# B&R Automation Studio project NAEUL004C00R13L518F00 (part 9)

#### Act_Main_P0200.st
```iecst
(** 2018-12-21 **)
ACTION Act_Main_P0200:
		//Conveyor Direction - SMEMA Arrow Indicator
	IF p_tyNtParamCurr.bUIConvDirRL THEN
		fUIInRtStatHide(ADR(tyP0200OpsGen.tyOps.tyBitmapUSIn.uiRtStat));
		fUIInRtStatHide(ADR(tyP0200OpsGen.tyOps.tyBitmapUSOut.uiRtStat));
		fUIInRtStatHide(ADR(tyP0200OpsGen.tyOps.tyTxtLane.uiRtStat));
		fUIInRtStatHide(ADR(tyP0200OpsGen.tyOps.tyHotspotUSAVSMEMA.uiRtStat));
		fUIInRtStatHide(ADR(tyP0200OpsGen.tyOps.tyBitmapUSAComm.uiRtStat));
		fUIInRtStatHide(ADR(tyP0200OpsGen.tyOps.tyBitmapUSAComm.uiMaskRtStat));

		fUIInRtStatHide(ADR(tyP0200OpsGen.tyUSCommB.tyBitmapUSIn.uiRtStat));
		fUIInRtStatHide(ADR(tyP0200OpsGen.tyUSCommB.tyBitmapUSOut.uiRtStat));
		fUIInRtStatHide(ADR(tyP0200OpsGen.tyUSCommB.tyTxtLane.uiRtStat));
		fUIInRtStatHide(ADR(tyP0200OpsGen.tyUSCommB.tyHotspotUSBVSMEMA.uiRtStat));
		fUIInRtStatHide(ADR(tyP0200OpsGen.tyUSCommB.tyBitmapUSBComm.uiRtStat));
		fUIInRtStatHide(ADR(tyP0200OpsGen.tyUSCommB.tyBitmapUSBComm.uiMaskRtStat));

		fUIInRtStatOff(ADR(tyP0200OpsGen.tyOps.tyBitmapUSIn1.uiRtStat));
		fUIInRtStatOff(ADR(tyP0200OpsGen.tyOps.tyBitmapUSOut1.uiRtStat));
		fUIInRtStatOff(ADR(tyP0200OpsGen.tyOps.tyTxtLane1.uiRtStat));
		//	fUIInRtStatOff(ADR(tyP0200OpsGen.tyOps.tyHotspotUSAVSMEMA1.uiRtStat));
		fUIInRtStatOff(ADR(tyP0200OpsGen.tyOps.tyBitmapUSAComm1.uiRtStat));
		fUIInRtStatOff(ADR(tyP0200OpsGen.tyOps.tyBitmapUSAComm1.uiMaskRtStat));

		fUIInRtStatOff(ADR(tyP0200OpsGen.tyUSCommB.tyBitmapUSIn1.uiRtStat));
		fUIInRtStatOff(ADR(tyP0200OpsGen.tyUSCommB.tyBitmapUSOut1.uiRtStat));
		fUIInRtStatOff(ADR(tyP0200OpsGen.tyUSCommB.tyTxtLane1.uiRtStat));
		//	fUIInRtStatOff(ADR(tyP0200OpsGen.tyUSCommB.tyHotspotUSBVSMEMA1.uiRtStat));
		fUIInRtStatOff(ADR(tyP0200OpsGen.tyUSCommB.tyBitmapUSBComm1.uiRtStat));
		fUIInRtStatOff(ADR(tyP0200OpsGen.tyUSCommB.tyBitmapUSBComm1.uiMaskRtStat));

	ELSE

		fUIInRtStatOff(ADR(tyP0200OpsGen.tyOps.tyBitmapUSIn.uiRtStat));
		fUIInRtStatOff(ADR(tyP0200OpsGen.tyOps.tyBitmapUSOut.uiRtStat));
		fUIInRtStatOff(ADR(tyP0200OpsGen.tyOps.tyTxtLane.uiRtStat));
		//		fUIInRtStatOff(ADR(tyP0200OpsGen.tyOps.tyHotspotUSAVSMEMA.uiRtStat));
		fUIInRtStatOff(ADR(tyP0200OpsGen.tyOps.tyBitmapUSAComm.uiRtStat));
		fUIInRtStatOff(ADR(tyP0200OpsGen.tyOps.tyBitmapUSAComm.uiMaskRtStat));

		fUIInRtStatOff(ADR(tyP0200OpsGen.tyUSCommB.tyBitmapUSIn.uiRtStat));
		fUIInRtStatOff(ADR(tyP0200OpsGen.tyUSCommB.tyBitmapUSOut.uiRtStat));
		fUIInRtStatOff(ADR(tyP0200OpsGen.tyUSCommB.tyTxtLane.uiRtStat));
		//	fUIInRtStatOff(ADR(tyP0200OpsGen.tyUSCommB.tyHotspotUSBVSMEMA.uiRtStat));
		fUIInRtStatOff(ADR(tyP0200OpsGen.tyUSCommB.tyBitmapUSBComm.uiRtStat));
		fUIInRtStatOff(ADR(tyP0200OpsGen.tyUSCommB.tyBitmapUSBComm.uiMaskRtStat));

		fUIInRtStatHide(ADR(tyP0200OpsGen.tyOps.tyBitmapUSIn1.uiRtStat));
		fUIInRtStatHide(ADR(tyP0200OpsGen.tyOps.tyBitmapUSOut1.uiRtStat));
		fUIInRtStatHide(ADR(tyP0200OpsGen.tyOps.tyTxtLane1.uiRtStat));
		fUIInRtStatHide(ADR(tyP0200OpsGen.tyOps.tyHotspotUSAVSMEMA1.uiRtStat));
		fUIInRtStatHide(ADR(tyP0200OpsGen.tyOps.tyBitmapUSAComm1.uiRtStat));
		fUIInRtStatHide(ADR(tyP0200OpsGen.tyOps.tyBitmapUSAComm1.uiMaskRtStat));

		fUIInRtStatHide(ADR(tyP0200OpsGen.tyUSCommB.tyBitmapUSIn1.uiRtStat));
		fUIInRtStatHide(ADR(tyP0200OpsGen.tyUSCommB.tyBitmapUSOut1.uiRtStat));
		fUIInRtStatHide(ADR(tyP0200OpsGen.tyUSCommB.tyTxtLane1.uiRtStat));
		fUIInRtStatHide(ADR(tyP0200OpsGen.tyUSCommB.tyHotspotUSBVSMEMA1.uiRtStat));
		fUIInRtStatHide(ADR(tyP0200OpsGen.tyUSCommB.tyBitmapUSBComm1.uiRtStat));
		fUIInRtStatHide(ADR(tyP0200OpsGen.tyUSCommB.tyBitmapUSBComm1.uiMaskRtStat));

	END_IF

	//Display L to R
	tyP0200OpsGen.tyOps.tyHotspotOpsMagInfo.uiRtStat.0	:= p_tyNtParamCurr.bUIConvDirRL = TRUE;

	tyP0200OpsGen.tyOps.tyTxtMag1Slt.uiRtStat.0 		:= p_tyNtParamCurr.bUIConvDirRL = TRUE;
	tyP0200OpsGen.tyOps.tyTxtMag1Backslash.uiRtStat.0	:= p_tyNtParamCurr.bUIConvDirRL = TRUE;
	tyP0200OpsGen.tyOps.tyNumMag1AvlQty.uiRtStat.0		:= p_tyNtParamCurr.bUIConvDirRL = TRUE;
	tyP0200OpsGen.tyOps.tyNumMag1TtlSlt.uiRtStat.0		:= p_tyNtParamCurr.bUIConvDirRL = TRUE;

	tyP0200OpsGen.tyOps.tyTxtMag2Slt.uiRtStat.0 		:= p_tyNtParamCurr.bUIConvDirRL = TRUE;
	tyP0200OpsGen.tyOps.tyTxtMag2Backslash.uiRtStat.0	:= p_tyNtParamCurr.bUIConvDirRL = TRUE;
	tyP0200OpsGen.tyOps.tyNumMag2AvlQty.uiRtStat.0		:= p_tyNtParamCurr.bUIConvDirRL = TRUE;
	tyP0200OpsGen.tyOps.tyNumMag2TtlSlt.uiRtStat.0		:= p_tyNtParamCurr.bUIConvDirRL = TRUE;

	tyP0200OpsGen.tyOps.tyTxtMag3Slt.uiRtStat.0		:= NOT(p_tyNtParamCurr.eProjMag = ULMagTriple) OR p_tyNtParamCurr.bUIConvDirRL = TRUE;
	tyP0200OpsGen.tyOps.tyTxtBackslash3.uiRtStat.0	:= NOT(p_tyNtParamCurr.eProjMag = ULMagTriple) OR p_tyNtParamCurr.bUIConvDirRL = TRUE;
	tyP0200OpsGen.tyOps.tyNumMag3AvlQty.uiRtStat.0	:= NOT(p_tyNtParamCurr.eProjMag = ULMagTriple) OR p_tyNtParamCurr.bUIConvDirRL = TRUE;
	tyP0200OpsGen.tyOps.tyNumMag3TtlSlt.uiRtStat.0	:= NOT(p_tyNtParamCurr.eProjMag = ULMagTriple) OR p_tyNtParamCurr.bUIConvDirRL = TRUE;

	tyP0200OpsGen.tyOps.tyHotspotOps2Mag1.uiRtStat.0	:= NOT(p_tyNtParamCurr.eProjMag = ULMagDual);
	tyP0200OpsGen.tyOps.tyHotspotOps2Mag2.uiRtStat.0	:= NOT(p_tyNtParamCurr.eProjMag = ULMagDual);
	tyP0200OpsGen.tyOps.tyHotspotOps3Mag1.uiRtStat.0	:= NOT(p_tyNtParamCurr.eProjMag = ULMagTriple);
	tyP0200OpsGen.tyOps.tyHotspotOps3Mag2.uiRtStat.0	:= NOT(p_tyNtParamCurr.eProjMag = ULMagTriple);
	tyP0200OpsGen.tyOps.tyHotspotOps3Mag3.uiRtStat.0	:= NOT(p_tyNtParamCurr.eProjMag = ULMagTriple);

	tyP0200OpsGen.tyOps.tyTxtMagSlt.uiRtStat.0			:= p_tyNtParamCurr.bUIConvDirRL = TRUE;
	tyP0200OpsGen.tyOps.tyTxtMagSltBackslash.uiRtStat.0	:= p_tyNtParamCurr.bUIConvDirRL = TRUE;
	tyP0200OpsGen.tyOps.tyNumMinSltRange.uiRtStat.0		:= p_tyNtParamCurr.bUIConvDirRL = TRUE;
	tyP0200OpsGen.tyOps.tyNumMaxSltRange.uiRtStat.0		:= p_tyNtParamCurr.bUIConvDirRL = TRUE;

	tyP0200OpsGen.tyOps.tyTxtPitchSlt.uiRtStat.0		:= p_tyNtParamCurr.bUIConvDirRL = TRUE;
	tyP0200OpsGen.tyOps.tyNumPitch.uiRtStat.0			:= p_tyNtParamCurr.bUIConvDirRL = TRUE;

	tyP0200OpsGen.tyOps.tyHotspotOvenGroup.uiRtStat.0		:= p_tyNtParamCurr.bUIConvDirRL = TRUE;

	//Display R to L
	tyP0200OpsGen.tyOps.tyHotspotOpsMagInfoRToL.uiRtStat.0	:= p_tyNtParamCurr.bUIConvDirRL = FALSE;

	tyP0200OpsGen.tyOps.tyTxtMag1SltRToL.uiRtStat.0 		:= p_tyNtParamCurr.bUIConvDirRL = FALSE;
	tyP0200OpsGen.tyOps.tyTxtMag1BackslashRToL.uiRtStat.0	:= p_tyNtParamCurr.bUIConvDirRL = FALSE;
	tyP0200OpsGen.tyOps.tyNumMag1AvlQtyRToL.uiRtStat.0		:= p_tyNtParamCurr.bUIConvDirRL = FALSE;
	tyP0200OpsGen.tyOps.tyNumMag1TtlSltRToL.uiRtStat.0		:= p_tyNtParamCurr.bUIConvDirRL = FALSE;

	tyP0200OpsGen.tyOps.tyTxtMag2SltRToL.uiRtStat.0 		:= p_tyNtParamCurr.bUIConvDirRL = FALSE;
	tyP0200OpsGen.tyOps.tyTxtMag2BackslashRToL.uiRtStat.0	:= p_tyNtParamCurr.bUIConvDirRL = FALSE;
	tyP0200OpsGen.tyOps.tyNumMag2AvlQtyRToL.uiRtStat.0		:= p_tyNtParamCurr.bUIConvDirRL = FALSE;
	tyP0200OpsGen.tyOps.tyNumMag2TtlSltRToL.uiRtStat.0		:= p_tyNtParamCurr.bUIConvDirRL = FALSE;

	tyP0200OpsGen.tyOps.tyTxtMag3SltRToL.uiRtStat.0			:= NOT(p_tyNtParamCurr.eProjMag = ULMagTriple) OR p_tyNtParamCurr.bUIConvDirRL = FALSE;
	tyP0200OpsGen.tyOps.tyTxtMag3BackslashRToL.uiRtStat.0	:= NOT(p_tyNtParamCurr.eProjMag = ULMagTriple) OR p_tyNtParamCurr.bUIConvDirRL = FALSE;
	tyP0200OpsGen.tyOps.tyNumMag3AvlQtyRToL.uiRtStat.0		:= NOT(p_tyNtParamCurr.eProjMag = ULMagTriple) OR p_tyNtParamCurr.bUIConvDirRL = FALSE;
	tyP0200OpsGen.tyOps.tyNumMag3TtlSltRToL.uiRtStat.0		:= NOT(p_tyNtParamCurr.eProjMag = ULMagTriple) OR p_tyNtParamCurr.bUIConvDirRL = FALSE;

	tyP0200OpsGen.tyOps.tyTxtMagSltRToL.uiRtStat.0			:= p_tyNtParamCurr.bUIConvDirRL = FALSE;
	tyP0200OpsGen.tyOps.tyTxtMagSltBackslashRToL.uiRtStat.0	:= p_tyNtParamCurr.bUIConvDirRL = FALSE;
	tyP0200OpsGen.tyOps.tyNumMinSltRangeRToL.uiRtStat.0		:= p_tyNtParamCurr.bUIConvDirRL = FALSE;
	tyP0200OpsGen.tyOps.tyNumMaxSltRangeRToL.uiRtStat.0		:= p_tyNtParamCurr.bUIConvDirRL = FALSE;

	tyP0200OpsGen.tyOps.tyTxtPitchSltRToL.uiRtStat.0		:= p_tyNtParamCurr.bUIConvDirRL = FALSE;
	tyP0200OpsGen.tyOps.tyNumPitchRToL.uiRtStat.0			:= p_tyNtParamCurr.bUIConvDirRL = FALSE;

	tyP0200OpsGen.tyOps.tyHotspotOvenGroupRL.uiRtStat.0		:= p_tyNtParamCurr.bUIConvDirRL = FALSE;

	//L to R
	tyP0200OpsGen.tyOps.tyHotspotOps2Mag1.uiRtStat.0	:= NOT(p_tyNtParamCurr.eProjMag = ULMagDual) OR p_tyNtParamCurr.bUIConvDirRL = TRUE;
	tyP0200OpsGen.tyOps.tyHotspotOps2Mag2.uiRtStat.0	:= NOT(p_tyNtParamCurr.eProjMag = ULMagDual)OR p_tyNtParamCurr.bUIConvDirRL = TRUE;
	tyP0200OpsGen.tyOps.tyHotspotOps3Mag1.uiRtStat.0	:= NOT(p_tyNtParamCurr.eProjMag = ULMagTriple)OR p_tyNtParamCurr.bUIConvDirRL = TRUE;
	tyP0200OpsGen.tyOps.tyHotspotOps3Mag2.uiRtStat.0	:= NOT(p_tyNtParamCurr.eProjMag = ULMagTriple)OR p_tyNtParamCurr.bUIConvDirRL = TRUE;
	tyP0200OpsGen.tyOps.tyHotspotOps3Mag3.uiRtStat.0	:= NOT(p_tyNtParamCurr.eProjMag = ULMagTriple)OR p_tyNtParamCurr.bUIConvDirRL = TRUE;
	tyP0200OpsGen.tyOps.tyHotspotOpsTravLifter.uiRtStat.0		:= p_tyNtParamCurr.bUIConvDirRL = TRUE;
	//R to L
	tyP0200OpsGen.tyOps.tyHotspotOps2Mag1RToL.uiRtStat.0	:= NOT(p_tyNtParamCurr.eProjMag = ULMagDual) OR p_tyNtParamCurr.bUIConvDirRL = FALSE;
	tyP0200OpsGen.tyOps.tyHotspotOps2Mag2RToL.uiRtStat.0	:= NOT(p_tyNtParamCurr.eProjMag = ULMagDual)OR p_tyNtParamCurr.bUIConvDirRL = FALSE;
	tyP0200OpsGen.tyOps.tyHotspotOps3Mag1RToL.uiRtStat.0	:= NOT(p_tyNtParamCurr.eProjMag = ULMagTriple)OR p_tyNtParamCurr.bUIConvDirRL = FALSE;
	tyP0200OpsGen.tyOps.tyHotspotOps3Mag2RToL.uiRtStat.0	:= NOT(p_tyNtParamCurr.eProjMag = ULMagTriple)OR p_tyNtParamCurr.bUIConvDirRL = FALSE;
	tyP0200OpsGen.tyOps.tyHotspotOps3Mag3RToL.uiRtStat.0	:= NOT(p_tyNtParamCurr.eProjMag = ULMagTriple)OR p_tyNtParamCurr.bUIConvDirRL = FALSE;
	tyP0200OpsGen.tyOps.tyHotspotOpsTravRToL.uiRtStat.0		:= p_tyNtParamCurr.bUIConvDirRL = FALSE;

	//Oven
	tyP0200OpsGen.tyOven.tyTxtCntr.uiRtStat.0	:= NOT (p_tyNtParamCurr.bOvenInfoExtdPrep AND p_tyNtParamCurr.bUIConvDirRL);
	//tyP0200OpsGen.tyOven.tyTxtA.uiRtStat.0		:= p_tyNtParamCurr.bUIConvDirRL; //added
	tyP0200OpsGen.tyOven.tyTxtB.uiRtStat.0		:= NOT (p_tyNtParamCurr.bProjLaneBPrep AND p_tyNtParamCurr.bUIConvDirRL);
	//tyP0200OpsGen.tyOven.tyBtnOvenA.uiRtStat.0	:= p_tyNtParamCurr.bUIConvDirRL; //added
	tyP0200OpsGen.tyOven.tyBtnOvenB.uiRtStat.0	:= NOT (p_tyNtParamCurr.bProjLaneBPrep AND p_tyNtParamCurr.bUIConvDirRL);
	tyP0200OpsGen.tyOven.tyBtnCntrA.uiRtStat.0	:= NOT (p_tyNtParamCurr.bOvenInfoExtdPrep AND p_tyNtParamCurr.bUIConvDirRL);
	tyP0200OpsGen.tyOven.tyBtnCntrB.uiRtStat.0	:= NOT(p_tyNtParamCurr.bOvenInfoExtdPrep AND p_tyNtParamCurr.bProjLaneBPrep AND p_tyNtParamCurr.bUIConvDirRL);
	//R to L
	tyP0200OpsGen.tyOven.tyTxtCntrRToL.uiRtStat.0	:= NOT (p_tyNtParamCurr.bOvenInfoExtdPrep AND p_tyNtParamCurr.bUIConvDirRL = FALSE);
	tyP0200OpsGen.tyOven.tyTxtBRToL.uiRtStat.0		:= NOT (p_tyNtParamCurr.bProjLaneBPrep AND p_tyNtParamCurr.bUIConvDirRL = FALSE);
	tyP0200OpsGen.tyOven.tyBtnOvenBRToL.uiRtStat.0	:= NOT (p_tyNtParamCurr.bProjLaneBPrep AND p_tyNtParamCurr.bUIConvDirRL = FALSE);
	tyP0200OpsGen.tyOven.tyBtnCntrARToL.uiRtStat.0	:= NOT (p_tyNtParamCurr.bOvenInfoExtdPrep AND p_tyNtParamCurr.bUIConvDirRL = FALSE);
	tyP0200OpsGen.tyOven.tyBtnCntrBRToL.uiRtStat.0	:= NOT(p_tyNtParamCurr.bOvenInfoExtdPrep AND p_tyNtParamCurr.bProjLaneBPrep AND p_tyNtParamCurr.bUIConvDirRL = FALSE);

	//Machine Bitmap
	IF p_tyNtParamCurr.eProjMag = ULMagTriple THEN
		IF p_tyNtParamCurr.bProjLifterMagPlatform AND p_tyNtParamCurr.bUIConvDirRL THEN
			tyP0200OpsGen.tyOps.tyBitmapMc.uiValueIdx	:= 800;
		ELSIF p_tyNtParamCurr.bProjLifterMagPlatform THEN
			tyP0200OpsGen.tyOps.tyBitmapMc.uiValueIdx	:= 500;
		ELSIF p_tyNtParamCurr.bMagAutoVerifyPrep = FALSE THEN
			tyP0200OpsGen.tyOps.tyBitmapMc.uiValueIdx	:= 100;
		ELSE
			tyP0200OpsGen.tyOps.tyBitmapMc.uiValueIdx	:= 200; //200
		END_IF
	ELSIF p_tyNtParamCurr.eProjMag = ULMagDual THEN
		IF p_tyNtParamCurr.bProjLifterMagPlatform AND p_tyNtParamCurr.bUIConvDirRL THEN
			tyP0200OpsGen.tyOps.tyBitmapMc.uiValueIdx	:= 700;
		ELSIF p_tyNtParamCurr.bProjLifterMagPlatform AND p_tyNtParamCurr.bUIConvDirRL = FALSE AND p_tyNtParamCurr.bProjMagConvLane1Prep THEN
			tyP0200OpsGen.tyOps.tyBitmapMc.uiValueIdx	:= 900;
		ELSIF p_tyNtParamCurr.bProjLifterMagPlatform THEN
			tyP0200OpsGen.tyOps.tyBitmapMc.uiValueIdx	:= 600;
		ELSIF p_tyNtParamCurr.bMagAutoVerifyPrep = FALSE THEN
			tyP0200OpsGen.tyOps.tyBitmapMc.uiValueIdx	:= 300;
		ELSE
			tyP0200OpsGen.tyOps.tyBitmapMc.uiValueIdx	:= 300;
		END_IF
	END_IF

	//Communication
	tyP0200OpsGen.tyUSCommB.tyLyr.uiRtStat.0 := NOT(p_tyNtParamCurr.bProjLaneBPrep);

	//Direction
	CASE p_tyNtParamCurr.eProjConvDir OF
		ConvDirLToR:
			tyP0200OpsGen.tyOps.tyBitmapDir1.usiValueIdx	:= 0;	// -->>
			tyP0200OpsGen.tyOps.tyBitmapDir2.usiValueIdx	:= 0;	// -->>
		ConvDirRToL:
			tyP0200OpsGen.tyOps.tyBitmapDir1.usiValueIdx	:= 1;	// <<--
			tyP0200OpsGen.tyOps.tyBitmapDir2.usiValueIdx	:= 1;	// <<--
	END_CASE

	//Hide Warning Bitmap for LF
//	fUIInRtStatHide(ADR(tyP0200OpsGen.tyOps.tyTxtLdrInActiveCtrl.uiRtStat));
//	fUIInRtStatHide(ADR(tyP0201OpsTravLifter.tyOps.tyTxtLdrInActiveCtrl.uiRtStat));
//	fUIInRtStatHide(ADR(tyP0202OpsMag1.tyOps.tyTxtLdrInActiveCtrl.uiRtStat));
//	fUIInRtStatHide(ADR(tyP0203OpsMag2.tyOps.tyTxtLdrInActiveCtrl.uiRtStat));
//	fUIInRtStatHide(ADR(tyP0204OpsMag3.tyOps.tyTxtLdrInActiveCtrl.uiRtStat));
//
//	fUIInRtStatHide(ADR(tyP0200OpsGen.tyOps.tyBitmapWarningLF.uiRtStat));
//	fUIInRtStatHide(ADR(tyP0201OpsTrav.tyOps.tyBitmapWarningLF.uiRtStat));
//	fUIInRtStatHide(ADR(tyP0202OpsMag1.tyOps.tyBitmapWarningLF.uiRtStat));
//	fUIInRtStatHide(ADR(tyP0203OpsMag2.tyOps.tyBitmapWarningLF.uiRtStat));
	//	fUIInRtStatHide(ADR(tyP0204OpsMag3.tyOps.tyBitmapWarningLF.uiRtStat));

	tyP0200OpsGen.tyOps.tyHotspotOpsAIV.uiRtStat.0 := NOT(p_tyNtParamCurr.bProjAGVPrep AND p_tyNtParamCurr.bProjTCPAGVSigPrep);
	tyP0200OpsGen.tyOps.tyHotspotOpsAIV.uiMaskRtStat.0 := NOT(p_tyNtParamCurr.bProjAGVPrep AND p_tyNtParamCurr.bProjTCPAGVSigPrep);
	tyP0200OpsGen.tyOps.tyHotspotAIVGroup1.uiRtStat.0 := p_tyNtParamCurr.bProjMagConvLane1Prep = TRUE AND p_tyNtParamCurr.bProjAGVPrep; //left pic
	tyP0200OpsGen.tyOps.tyHotspotAIVGroup.uiRtStat.0 := p_tyNtParamCurr.bProjMagConvLane1Prep = FALSE AND NOT(p_tyNtParamCurr.bProjAGVPrep); //right pic

	tyP0200OpsGen.tyOps.tyHotspotOpsMagLane1.uiRtStat := NOT(p_tyNtParamCurr.bProjMagConvLane1Prep);
	tyP0200OpsGen.tyOps.tyHotspotOpsMagLane2.uiRtStat := NOT(p_tyNtParamCurr.bProjMagConvLane2Prep);

END_ACTION
```

#### Act_Main_P0201.st
```iecst
(** 2018-12-21 **)
ACTION Act_Main_P0201:

	//Display
	IF p_tyNtParamCurr.bProjLaneBPrep = FALSE THEN
		fUIInRtStatHide(ADR(tyP0201OpsTravLifter.tyIOMonitor.tyBtnUBAB.uiRtStat));
		fUIInRtStatHide(ADR(tyP0201OpsTravLifter.tyIOMonitor.tyBtnUBABStat.uiRtStat));
		fUIInRtStatHide(ADR(tyP0201OpsTravLifter.tyIOMonitor.tyBtnOvenInfeedSigB.uiRtStat));

		fUIInRtStatHide(ADR(tyP0201OpsTravLifter.tyIOMonitor.tyBtnUSBB.uiRtStat));
		fUIInRtStatHide(ADR(tyP0201OpsTravLifter.tyIOMonitor.tyBtnOvenInfoSigB.uiRtStat));
		fUIInRtStatHide(ADR(tyP0201OpsTravLifter.tyIOMonitor.tyBtnStopperUnBlkCtrlB.uiRtStat));
	END_IF

	IF p_tyNtParamCurr.bOvenInfoExtdPrep = FALSE THEN
		fUIInRtStatHide(ADR(tyP0201OpsTravLifter.tyIOMonitor.tyBtnOvenInfeedSigA.uiRtStat));
		fUIInRtStatHide(ADR(tyP0201OpsTravLifter.tyIOMonitor.tyBtnOvenInfeedSigB.uiRtStat));
	END_IF

	IF p_tyNtParamCurr.bProjInletShutPrep = FALSE THEN
		fUIInRtStatHide(ADR(tyP0201OpsTravLifter.tyIOMonitor.tyBtnInletShutterCloseSen.uiRtStat));
		fUIInRtStatHide(ADR(tyP0201OpsTravLifter.tyIOMonitor.tyBtnInletShutterOpenSen.uiRtStat));

		fUIInRtStatHide(ADR(tyP0201OpsTravLifter.tyIOMonitor.tyBtnInShutterCloseCtrl.uiRtStat));
		fUIInRtStatHide(ADR(tyP0201OpsTravLifter.tyIOMonitor.tyBtnInShutterOpenCtrl.uiRtStat));
	END_IF

	IF p_tyNtParamCurr.bProjOutletShutPrep = FALSE THEN
		fUIInRtStatHide(ADR(tyP0201OpsTravLifter.tyIOMonitor.tyBtnOutletShutterCloseSen.uiRtStat));
		fUIInRtStatHide(ADR(tyP0201OpsTravLifter.tyIOMonitor.tyBtnOutletShutterOpenSen.uiRtStat));
		fUIInRtStatHide(ADR(tyP0201OpsTravLifter.tyIOMonitor.tyBtnOutShutterCloseCtrl.uiRtStat));
		fUIInRtStatHide(ADR(tyP0201OpsTravLifter.tyIOMonitor.tyBtnOutShutterOpenCtrl.uiRtStat));
	END_IF
	IF p_tyNtParamCurr.bProjOutletShut2Prep = FALSE THEN
		fUIInRtStatHide(ADR(tyP0201OpsTravLifter.tyIOMonitor.tyBtnOutletShutterCloseSen2.uiRtStat));
		fUIInRtStatHide(ADR(tyP0201OpsTravLifter.tyIOMonitor.tyBtnOutletShutterOpenSen2.uiRtStat));
		fUIInRtStatHide(ADR(tyP0201OpsTravLifter.tyIOMonitor.tyBtnOutShutterCloseCtrl2.uiRtStat));
		fUIInRtStatHide(ADR(tyP0201OpsTravLifter.tyIOMonitor.tyBtnOutShutterOpenCtrl2.uiRtStat));
	END_IF
	IF p_tyNtParamCurr.bProjOutletShut3Prep = FALSE THEN
		fUIInRtStatHide(ADR(tyP0201OpsTravLifter.tyIOMonitor.tyBtnOutletShutterCloseSen3.uiRtStat));
		fUIInRtStatHide(ADR(tyP0201OpsTravLifter.tyIOMonitor.tyBtnOutletShutterOpenSen3.uiRtStat));
		fUIInRtStatHide(ADR(tyP0201OpsTravLifter.tyIOMonitor.tyBtnOutShutterCloseCtrl3.uiRtStat));
		fUIInRtStatHide(ADR(tyP0201OpsTravLifter.tyIOMonitor.tyBtnOutShutterOpenCtrl3.uiRtStat));
	END_IF
	//Change Parameter
	IF p_tyNtParamCurr.bProjLaneBPrep THEN
		tyP0201OpsTravLifter.tyParam.tyDrpDnMcMode.usiValueMaxIdx	:= 8;
	ELSE
		tyP0201OpsTravLifter.tyParam.tyDrpDnMcMode.usiValueMaxIdx	:= 2;
	END_IF

	//Digital Input Used
	IF p_tyNtParamCurr.tyDISettings.diSafetyRlySig = 0 THEN
		fUIInRtStatHide(ADR(tyP0201OpsTravLifter.tyIOMonitor.tyBtnSafetyRlySig.uiRtStat));
	END_IF

	IF p_tyNtParamCurr.tyDISettings.diEStopSig = 0 THEN
		fUIInRtStatHide(ADR(tyP0201OpsTravLifter.tyIOMonitor.tyBtnEStop.uiRtStat));
	END_IF

	IF p_tyNtParamCurr.tyDISettings.diCoverSWSig = 0 THEN
		fUIInRtStatHide(ADR(tyP0201OpsTravLifter.tyIOMonitor.tyBtnCoverSWSig.uiRtStat));
	END_IF

	IF p_tyNtParamCurr.tyDISettings.diUBAA = 0 THEN
		fUIInRtStatHide(ADR(tyP0201OpsTravLifter.tyIOMonitor.tyBtnUBAA.uiRtStat));
	END_IF

	IF p_tyNtParamCurr.tyDISettings.diUBAAStat = 0 THEN
		fUIInRtStatHide(ADR(tyP0201OpsTravLifter.tyIOMonitor.tyBtnUBAAStat.uiRtStat));
	END_IF

	IF p_tyNtParamCurr.tyDISettings.diUBAB = 0 THEN
		fUIInRtStatHide(ADR(tyP0201OpsTravLifter.tyIOMonitor.tyBtnUBAB.uiRtStat));
	END_IF

	IF p_tyNtParamCurr.tyDISettings.diUBABStat = 0 THEN
		fUIInRtStatHide(ADR(tyP0201OpsTravLifter.tyIOMonitor.tyBtnUBABStat.uiRtStat));
	END_IF

	IF p_tyNtParamCurr.tyDISettings.diOvenInfeedSigA = 0 THEN
		fUIInRtStatHide(ADR(tyP0201OpsTravLifter.tyIOMonitor.tyBtnOvenInfeedSigA.uiRtStat));
	END_IF

	IF p_tyNtParamCurr.tyDISettings.diOvenInfeedSigB = 0 THEN
		fUIInRtStatHide(ADR(tyP0201OpsTravLifter.tyIOMonitor.tyBtnOvenInfeedSigB.uiRtStat));
	END_IF

	IF p_tyNtParamCurr.tyDISettings.diPusherExtRS = 0 THEN
		fUIInRtStatHide(ADR(tyP0201OpsTravLifter.tyIOMonitor.tyBtnPshrExtRS.uiRtStat));
	END_IF

	IF p_tyNtParamCurr.tyDISettings.diPusherRetRS = 0 THEN
		fUIInRtStatHide(ADR(tyP0201OpsTravLifter.tyIOMonitor.tyBtnPshrRetRS.uiRtStat));
	END_IF

	IF p_tyNtParamCurr.tyDISettings.diConvLftSen = 0 THEN
		fUIInRtStatHide(ADR(tyP0201OpsTravLifter.tyIOMonitor.tyBtnConvLftSen.uiRtStat));
	END_IF

	IF p_tyNtParamCurr.tyDISettings.diConvRgtSen = 0 THEN
		fUIInRtStatHide(ADR(tyP0201OpsTravLifter.tyIOMonitor.tyBtnConvRgtSen.uiRtStat));
	END_IF

	IF p_tyNtParamCurr.tyDISettings.diConvMidSen = 0 THEN
		fUIInRtStatHide(ADR(tyP0201OpsTravLifter.tyIOMonitor.tyBtnConvMidSen.uiRtStat));
	END_IF

	IF p_tyNtParamCurr.tyDISettings.diConvClrSen = 0 THEN
		fUIInRtStatHide(ADR(tyP0201OpsTravLifter.tyIOMonitor.tyBtnConvClrSen.uiRtStat));
	END_IF

	IF p_tyNtParamCurr.tyDISettings.diLifterTimingBeltSen = 0 THEN
		fUIInRtStatHide(ADR(tyP0201OpsTravLifter.tyIOMonitor.tyBtnLifterTmBeltSen.uiRtStat));
	END_IF

	IF p_tyNtParamCurr.tyDISettings.diInShutterOpenRS = 0 THEN
		fUIInRtStatHide(ADR(tyP0201OpsTravLifter.tyIOMonitor.tyBtnInletShutterOpenSen.uiRtStat));
	END_IF

	IF p_tyNtParamCurr.tyDISettings.diInShutterCloseRS = 0 THEN
		fUIInRtStatHide(ADR(tyP0201OpsTravLifter.tyIOMonitor.tyBtnInletShutterCloseSen.uiRtStat));
	END_IF

	IF p_tyNtParamCurr.tyDISettings.diOutShutterOpenRS = 0 THEN
		fUIInRtStatHide(ADR(tyP0201OpsTravLifter.tyIOMonitor.tyBtnOutletShutterOpenSen.uiRtStat));
	END_IF

	IF p_tyNtParamCurr.tyDISettings.diOutShutterCloseRS = 0 THEN
		fUIInRtStatHide(ADR(tyP0201OpsTravLifter.tyIOMonitor.tyBtnOutletShutterCloseSen.uiRtStat));
	END_IF

	IF p_tyNtParamCurr.tyDISettings.diOutShutterCloseRS2 = 0 THEN
		fUIInRtStatHide(ADR(tyP0201OpsTravLifter.tyIOMonitor.tyBtnOutletShutterCloseSen2.uiRtStat));
	END_IF

	IF p_tyNtParamCurr.tyDISettings.diOutShutterCloseRS3 = 0 THEN
		fUIInRtStatHide(ADR(tyP0201OpsTravLifter.tyIOMonitor.tyBtnOutletShutterCloseSen3.uiRtStat));
	END_IF
	IF p_tyNtParamCurr.tyDISettings.diPshrAntiJam = 0 THEN
		fUIInRtStatHide(ADR(tyP0201OpsTravLifter.tyIOMonitor.tyBtnAntiJamSen.uiRtStat));
	END_IF

	IF p_tyNtParamCurr.tyDISettings.diMagWidthChkSen = 0 THEN
		fUIInRtStatHide(ADR(tyP0201OpsTravLifter.tyIOMonitor.tyBtnMagWidthChk.uiRtStat));
	END_IF

	IF p_tyNtParamCurr.tyDISettings.diInletStopperASen = 0 THEN
		fUIInRtStatHide(ADR(tyP0201OpsTravLifter.tyIOMonitor.tyBtnInletStopperASensor.uiRtStat));
	END_IF

	IF p_tyNtParamCurr.tyDISettings.diScanComplSig = 0 THEN
		fUIInRtStatHide(ADR(tyP0201OpsTravLifter.tyIOMonitor1.tyBtnScannerComplSig.uiRtStat));
	END_IF
	IF p_tyNtParamCurr.tyDISettings.diPCBScanSen = 0 THEN
		fUIInRtStatHide(ADR(tyP0201OpsTravLifter.tyIOMonitor1.tyBtnPCBPresentSen.uiRtStat));
	END_IF

	//Digital Output Selected
	IF p_tyNtParamCurr.tyDOSettings.diSafetyRlyRst = 0 THEN
		fUIInRtStatHide(ADR(tyP0201OpsTravLifter.tyIOMonitor.tyBtnSafetyRlyRst.uiRtStat));
	END_IF

	IF p_tyNtParamCurr.tyDOSettings.diTLGreen = 0 THEN
		fUIInRtStatHide(ADR(tyP0201OpsTravLifter.tyIOMonitor.tyBtnTLGreen.uiRtStat));
	END_IF

	IF p_tyNtParamCurr.tyDOSettings.diTLAmber = 0 THEN
		fUIInRtStatHide(ADR(tyP0201OpsTravLifter.tyIOMonitor.tyBtnTLAmber.uiRtStat));
	END_IF

	IF p_tyNtParamCurr.tyDOSettings.diTLRed = 0 THEN
		fUIInRtStatHide(ADR(tyP0201OpsTravLifter.tyIOMonitor.tyBtnTLRed.uiRtStat));
	END_IF

	IF p_tyNtParamCurr.tyDOSettings.diBuzzer = 0 THEN
		fUIInRtStatHide(ADR(tyP0201OpsTravLifter.tyIOMonitor.tyBtnBuzzer.uiRtStat));
	END_IF

	IF p_tyNtParamCurr.tyDOSettings.diUSBA = 0 THEN
		fUIInRtStatHide(ADR(tyP0201OpsTravLifter.tyIOMonitor.tyBtnUSBA.uiRtStat));
	END_IF

	IF p_tyNtParamCurr.tyDOSettings.diUSBB = 0 THEN
		fUIInRtStatHide(ADR(tyP0201OpsTravLifter.tyIOMonitor.tyBtnUSBB.uiRtStat));
	END_IF

	IF p_tyNtParamCurr.tyDOSettings.diOvenInfoSigA = 0 THEN
		fUIInRtStatHide(ADR(tyP0201OpsTravLifter.tyIOMonitor.tyBtnOvenInfoSigA.uiRtStat));
	END_IF

	IF p_tyNtParamCurr.tyDOSettings.diOvenInfoSigB = 0 THEN
		fUIInRtStatHide(ADR(tyP0201OpsTravLifter.tyIOMonitor.tyBtnOvenInfoSigB.uiRtStat));
	END_IF

	IF p_tyNtParamCurr.tyDOSettings.diPusherExtCtrl = 0 THEN
		fUIInRtStatHide(ADR(tyP0201OpsTravLifter.tyIOMonitor.tyBtnPshrExtCtrl.uiRtStat));
	END_IF

	IF p_tyNtParamCurr.tyDOSettings.diStopperUnblkCtrlA = 0 THEN
		fUIInRtStatHide(ADR(tyP0201OpsTravLifter.tyIOMonitor.tyBtnStopperUnBlkCtrlA.uiRtStat));
	END_IF

	IF p_tyNtParamCurr.tyDOSettings.diStopperUnblkCtrlB = 0 THEN
		fUIInRtStatHide(ADR(tyP0201OpsTravLifter.tyIOMonitor.tyBtnStopperUnBlkCtrlB.uiRtStat));
	END_IF

	IF p_tyNtParamCurr.tyDOSettings.diInShutterOpenCtrl = 0 THEN
		fUIInRtStatHide(ADR(tyP0201OpsTravLifter.tyIOMonitor.tyBtnInShutterOpenCtrl.uiRtStat));
	END_IF

	IF p_tyNtParamCurr.tyDOSettings.diInShutterCloseCtrl = 0 THEN
		fUIInRtStatHide(ADR(tyP0201OpsTravLifter.tyIOMonitor.tyBtnInShutterCloseCtrl.uiRtStat));
	END_IF

	IF p_tyNtParamCurr.tyDOSettings.diOutShutterOpenCtrl = 0 THEN
		fUIInRtStatHide(ADR(tyP0201OpsTravLifter.tyIOMonitor.tyBtnOutShutterOpenCtrl.uiRtStat));
	END_IF

	IF p_tyNtParamCurr.tyDOSettings.diOutShutterCloseCtrl = 0 THEN
		fUIInRtStatHide(ADR(tyP0201OpsTravLifter.tyIOMonitor.tyBtnOutShutterCloseCtrl.uiRtStat));
	END_IF

	IF p_tyNtParamCurr.tyDOSettings.diOutShutterCloseCtrl2 = 0 THEN
		fUIInRtStatHide(ADR(tyP0201OpsTravLifter.tyIOMonitor.tyBtnOutShutterCloseCtrl2.uiRtStat));
	END_IF

	IF p_tyNtParamCurr.tyDOSettings.diOutShutterCloseCtrl3 = 0 THEN
		fUIInRtStatHide(ADR(tyP0201OpsTravLifter.tyIOMonitor.tyBtnOutShutterCloseCtrl3.uiRtStat));
	END_IF

	IF p_tyNtParamCurr.tyDOSettings.diPushConvMtrOn = 0 THEN
		fUIInRtStatHide(ADR(tyP0201OpsTravLifter.tyIOMonitor.tyBtnPshrMtrOn.uiRtStat));
	END_IF
	//scanner
	IF p_tyNtParamCurr.tyDOSettings.diScanTrigSig = 0 THEN
		fUIInRtStatHide(ADR(tyP0201OpsTravLifter.tyIOMonitor1.tyBtnTrigScannerSig.uiRtStat));
	END_IF
	IF p_tyNtParamCurr.tyDOSettings.diMag1ExitPCB = 0 THEN
		fUIInRtStatHide(ADR(tyP0201OpsTravLifter.tyIOMonitor1.tyBtnPCBExitMag1.uiRtStat));
	END_IF
	IF p_tyNtParamCurr.tyDOSettings.diMag2ExitPCB = 0 THEN
		fUIInRtStatHide(ADR(tyP0201OpsTravLifter.tyIOMonitor1.tyBtnPCBExitMag2.uiRtStat));
	END_IF
	IF p_tyNtParamCurr.tyDOSettings.diMag3ExitPCB = 0 THEN
		fUIInRtStatHide(ADR(tyP0201OpsTravLifter.tyIOMonitor1.tyBtnPCBExitMag3.uiRtStat));
	END_IF
	IF p_tyNtParamCurr.tyDOSettings.diScanTrigSig <> 0
		OR p_tyNtParamCurr.tyDOSettings.diMag1ExitPCB <> 0
		OR p_tyNtParamCurr.tyDOSettings.diMag2ExitPCB <> 0
		OR p_tyNtParamCurr.tyDOSettings.diMag3ExitPCB <> 0
		OR p_tyNtParamCurr.tyDISettings.diPCBScanSen <> 0
		OR p_tyNtParamCurr.tyDISettings.diScanComplSig <> 0 THEN
		bUITravLifShowIOMonitor2 := TRUE;
	END_IF

	IF p_tyNtParamCurr.eProjMag = ULMagTriple THEN
		IF p_tyNtParamCurr.bProjLifterMagPlatform AND p_tyNtParamCurr.bUIConvDirRL THEN
			tyP0201OpsTravLifter.tyOps.tyBitmapMc.uiValueIdx	:= 800;
		ELSIF p_tyNtParamCurr.bProjLifterMagPlatform THEN
			tyP0201OpsTravLifter.tyOps.tyBitmapMc.uiValueIdx	:= 500;
		ELSE
			tyP0201OpsTravLifter.tyOps.tyBitmapMc.uiValueIdx	:= 200; //Replace with 293
		END_IF
	ELSIF p_tyNtParamCurr.eProjMag = ULMagDual THEN
		IF p_tyNtParamCurr.bProjLifterMagPlatform AND p_tyNtParamCurr.bUIConvDirRL THEN
			tyP0201OpsTravLifter.tyOps.tyBitmapMc.uiValueIdx	:= 700;
		ELSIF p_tyNtParamCurr.bProjLifterMagPlatform AND p_tyNtParamCurr.bUIConvDirRL = FALSE AND p_tyNtParamCurr.bProjMagConvLane1Prep THEN
			tyP0201OpsTravLifter.tyOps.tyBitmapMc.uiValueIdx	:= 900;
		ELSIF p_tyNtParamCurr.bProjLifterMagPlatform THEN
			tyP0201OpsTravLifter.tyOps.tyBitmapMc.uiValueIdx	:= 600;
		ELSE
			tyP0201OpsTravLifter.tyOps.tyBitmapMc.uiValueIdx	:= 300;
		END_IF
	END_IF

	tyP0201OpsTravLifter.tyOps.tyNumMtrPshrExtSpd.uiRtStat.0	:= NOT p_tyNtParamCurr.bProjMotorizedPusherPrep;
	tyP0201OpsTravLifter.tyOps.tyNumMtrPshrExtTorq.uiRtStat.0	:= NOT p_tyNtParamCurr.bProjMotorizedPusherPrep;
	tyP0201OpsTravLifter.tyOps.tyNumPshrOffset.uiRtStat.0		:= NOT p_tyNtParamCurr.bProjMotorizedPusherPrep;

	IF p_tyNtParamCurr.eCustomerReq = Siemens THEN //Siemen
		tyP0201OpsTravLifter.tyIOMonitor.tyBtnTLAmber.usiTxtIdx := 25;
	END_IF

END_ACTION
```

#### Act_Main_P0202.st
```iecst
(** 2018-12-21 **)
ACTION Act_Main_P0202:

	//Machine Bitmap
	IF p_tyNtParamCurr.eProjMag = ULMagTriple THEN
		IF p_tyNtParamCurr.bProjLifterMagPlatform AND p_tyNtParamCurr.bUIConvDirRL THEN
			tyP0202OpsMag1.tyOps.tyBitmapMc.uiValueIdx	:= 800;
		ELSIF p_tyNtParamCurr.bProjLifterMagPlatform THEN
			tyP0202OpsMag1.tyOps.tyBitmapMc.uiValueIdx	:= 500;
		ELSE
			tyP0202OpsMag1.tyOps.tyBitmapMc.uiValueIdx	:= 200;
		END_IF
	ELSIF p_tyNtParamCurr.eProjMag = ULMagDual THEN
		IF p_tyNtParamCurr.bProjLifterMagPlatform AND p_tyNtParamCurr.bUIConvDirRL THEN
			tyP0202OpsMag1.tyOps.tyBitmapMc.uiValueIdx	:= 700;
		ELSIF p_tyNtParamCurr.bProjLifterMagPlatform AND p_tyNtParamCurr.bUIConvDirRL = FALSE AND p_tyNtParamCurr.bProjMagConvLane1Prep THEN
			tyP0202OpsMag1.tyOps.tyBitmapMc.uiValueIdx	:= 900;
		ELSIF p_tyNtParamCurr.bProjLifterMagPlatform THEN
			tyP0202OpsMag1.tyOps.tyBitmapMc.uiValueIdx	:= 600;
		ELSE
			tyP0202OpsMag1.tyOps.tyBitmapMc.uiValueIdx	:= 300;
		END_IF
	END_IF

	//AIV
	//tyP0202OpsMag1.tyOps.tyTxtLblAIV.uiRtStat.0		:= NOT p_tyNtParamCurr.bProjAGVPrep;
	//tyP0202OpsMag1.tyOps.tyBtnAIVWifi.uiRtStat.0	:= NOT p_tyNtParamCurr.bProjAGVPrep;

	tyP0202OpsMag1.tyOps.tyTxtLblAIV.uiRtStat.0		:= TRUE;
	tyP0202OpsMag1.tyOps.tyBtnAIVWifi.uiRtStat.0	:= TRUE;
	//tyP0202OpsMag1.tyOps.tyBtnChgMag.uiRtStat.0	:= NOT(p_tyNtParamCurr.bProjBtnInsertRmvMag);
	//tyP0202OpsMag1.tyOps.tyBitmapChgMag.uiRtStat.0:= NOT(p_tyNtParamCurr.bProjBtnInsertRmvMag);
	tyP0202OpsMag1.tyOps.tyBtnChgMag.uiRtStat.0		:= NOT(p_tyNtParamCurr.bProjAGVPrep AND p_tyNtParamCurr.bProjBtnInsertRmvMag);
	tyP0202OpsMag1.tyOps.tyBitmapChgMag.uiRtStat.0	:= NOT(p_tyNtParamCurr.bProjAGVPrep AND p_tyNtParamCurr.bProjBtnInsertRmvMag);

	//Display
	IF p_tyNtParamCurr.bProjLaneBPrep = FALSE THEN
		fUIInRtStatHide(ADR(tyP0202OpsMag1.tyIOMonitor.tyBtnUBAB.uiRtStat));
		fUIInRtStatHide(ADR(tyP0202OpsMag1.tyIOMonitor.tyBtnUBABStat.uiRtStat));
		fUIInRtStatHide(ADR(tyP0202OpsMag1.tyIOMonitor.tyBtnOvenInfeedSigB.uiRtStat));

		fUIInRtStatHide(ADR(tyP0202OpsMag1.tyIOMonitor.tyBtnUSBB.uiRtStat));
		fUIInRtStatHide(ADR(tyP0202OpsMag1.tyIOMonitor.tyBtnOvenInfoSigB.uiRtStat));
	END_IF

	IF p_tyNtParamCurr.bOvenInfoExtdPrep = FALSE THEN
		fUIInRtStatHide(ADR(tyP0202OpsMag1.tyIOMonitor.tyBtnOvenInfeedSigA.uiRtStat));
		fUIInRtStatHide(ADR(tyP0202OpsMag1.tyIOMonitor.tyBtnOvenInfeedSigB.uiRtStat));
	END_IF

	//Change Parameter
	IF p_tyNtParamCurr.bProjLaneBPrep THEN
		tyP0202OpsMag1.tyParam.tyDrpDnMcMode.usiValueMaxIdx	:= 8;
	ELSE
		tyP0202OpsMag1.tyParam.tyDrpDnMcMode.usiValueMaxIdx	:= 2;
	END_IF

	//Digital Input Used
	IF p_tyNtParamCurr.tyDISettings.diSafetyRlySig = 0 THEN
		fUIInRtStatHide(ADR(tyP0202OpsMag1.tyIOMonitor.tyBtnSafetyRlySig.uiRtStat));
	END_IF

	IF p_tyNtParamCurr.tyDISettings.diEStopSig = 0 THEN
		fUIInRtStatHide(ADR(tyP0202OpsMag1.tyIOMonitor.tyBtnEStop.uiRtStat));
	END_IF

	IF p_tyNtParamCurr.tyDISettings.diCoverSWSig = 0 THEN
		fUIInRtStatHide(ADR(tyP0202OpsMag1.tyIOMonitor.tyBtnCoverSWSig.uiRtStat));
	END_IF

	IF p_tyNtParamCurr.tyDISettings.diUBAA = 0 THEN
		fUIInRtStatHide(ADR(tyP0202OpsMag1.tyIOMonitor.tyBtnUBAA.uiRtStat));
	END_IF

	IF p_tyNtParamCurr.tyDISettings.diUBAAStat = 0 THEN
		fUIInRtStatHide(ADR(tyP0202OpsMag1.tyIOMonitor.tyBtnUBAAStat.uiRtStat));
	END_IF

	IF p_tyNtParamCurr.tyDISettings.diUBAB = 0 THEN
		fUIInRtStatHide(ADR(tyP0202OpsMag1.tyIOMonitor.tyBtnUBAB.uiRtStat));
	END_IF

	IF p_tyNtParamCurr.tyDISettings.diUBABStat = 0 THEN
		fUIInRtStatHide(ADR(tyP0202OpsMag1.tyIOMonitor.tyBtnUBABStat.uiRtStat));
	END_IF

	IF p_tyNtParamCurr.tyDISettings.diOvenInfeedSigA = 0 THEN
		fUIInRtStatHide(ADR(tyP0202OpsMag1.tyIOMonitor.tyBtnOvenInfeedSigA.uiRtStat));
	END_IF

	IF p_tyNtParamCurr.tyDISettings.diOvenInfeedSigB = 0 THEN
		fUIInRtStatHide(ADR(tyP0202OpsMag1.tyIOMonitor.tyBtnOvenInfeedSigB.uiRtStat));
	END_IF

	IF p_tyNtParamCurr.tyDISettings.diMag1FixedClampRS = 0 THEN
		fUIInRtStatHide(ADR(tyP0202OpsMag1.tyIOMonitor.tyBtnMag1FixedClmpRS.uiRtStat));
	END_IF

	IF p_tyNtParamCurr.tyDISettings.diMag1FixedUnclampRS = 0 THEN
		fUIInRtStatHide(ADR(tyP0202OpsMag1.tyIOMonitor.tyBtnMag1FixedUnclmpRS.uiRtStat));
	END_IF

	IF p_tyNtParamCurr.tyDISettings.diMag1RemoteClampRS = 0 THEN
		fUIInRtStatHide(ADR(tyP0202OpsMag1.tyIOMonitor.tyBtnMag1RmtClmpRS.uiRtStat));
	END_IF

	IF p_tyNtParamCurr.tyDISettings.diMag1RemoteUnclampRS = 0 THEN
		fUIInRtStatHide(ADR(tyP0202OpsMag1.tyIOMonitor.tyBtnMag1RmtUnclmpRS.uiRtStat));
	END_IF

	IF p_tyNtParamCurr.tyDISettings.diMagConvEntSen1 = 0 THEN
		fUIInRtStatHide(ADR(tyP0202OpsMag1.tyIOMonitor.tyBtnMag1ConvEntrySen.uiRtStat));
	END_IF

	IF p_tyNtParamCurr.tyDISettings.diMagPresentSen1 = 0 THEN
		fUIInRtStatHide(ADR(tyP0202OpsMag1.tyIOMonitor.tyBtnMag1PresentSen.uiRtStat));
	END_IF

	IF p_tyNtParamCurr.tyDISettings.diMag1AIVInPosSen1 = 0 THEN
		fUIInRtStatHide(ADR(tyP0202OpsMag1.tyIOMonitor.tyBtnMag1AIVInPosSen1.uiRtStat));
	END_IF

	IF p_tyNtParamCurr.tyDISettings.diMag1AIVInPosSen2 = 0 THEN
		fUIInRtStatHide(ADR(tyP0202OpsMag1.tyIOMonitor.tyBtnMag1AIVInPosSen2.uiRtStat));
	END_IF

	IF p_tyNtParamCurr.tyDISettings.diMag1OrientChkSen1 = 0 THEN
		fUIInRtStatHide(ADR(tyP0202OpsMag1.tyIOMonitor.tyBtnMag1OrientationChkSen1.uiRtStat));
	END_IF

	IF p_tyNtParamCurr.tyDISettings.diMag1OrientChkSen2 = 0 THEN
		fUIInRtStatHide(ADR(tyP0202OpsMag1.tyIOMonitor.tyBtnMag1OrientationChkSen2.uiRtStat));
	END_IF

	//Digital Output Selected
	IF p_tyNtParamCurr.tyDOSettings.diSafetyRlyRst = 0 THEN
		fUIInRtStatHide(ADR(tyP0202OpsMag1.tyIOMonitor.tyBtnSafetyRlyRst.uiRtStat));
	END_IF

	IF p_tyNtParamCurr.tyDOSettings.diTLGreen = 0 THEN
		fUIInRtStatHide(ADR(tyP0202OpsMag1.tyIOMonitor.tyBtnTLGreen.uiRtStat));
	END_IF

	IF p_tyNtParamCurr.tyDOSettings.diTLAmber = 0 THEN
		fUIInRtStatHide(ADR(tyP0202OpsMag1.tyIOMonitor.tyBtnTLAmber.uiRtStat));
	END_IF

	IF p_tyNtParamCurr.tyDOSettings.diTLRed = 0 THEN
		fUIInRtStatHide(ADR(tyP0202OpsMag1.tyIOMonitor.tyBtnTLRed.uiRtStat));
	END_IF

	IF p_tyNtParamCurr.tyDOSettings.diBuzzer = 0 THEN
		fUIInRtStatHide(ADR(tyP0202OpsMag1.tyIOMonitor.tyBtnBuzzer.uiRtStat));
	END_IF

	IF p_tyNtParamCurr.tyDOSettings.diUSBA = 0 THEN
		fUIInRtStatHide(ADR(tyP0202OpsMag1.tyIOMonitor.tyBtnUSBA.uiRtStat));
	END_IF

	IF p_tyNtParamCurr.tyDOSettings.diUSBB = 0 THEN
		fUIInRtStatHide(ADR(tyP0202OpsMag1.tyIOMonitor.tyBtnUSBB.uiRtStat));
	END_IF

	IF p_tyNtParamCurr.tyDOSettings.diOvenInfoSigA = 0 THEN
		fUIInRtStatHide(ADR(tyP0202OpsMag1.tyIOMonitor.tyBtnOvenInfoSigA.uiRtStat));
	END_IF

	IF p_tyNtParamCurr.tyDOSettings.diOvenInfoSigB = 0 THEN
		fUIInRtStatHide(ADR(tyP0202OpsMag1.tyIOMonitor.tyBtnOvenInfoSigB.uiRtStat));
	END_IF

	IF p_tyNtParamCurr.tyDOSettings.diMag1FixedClampCtrl = 0 THEN
		fUIInRtStatHide(ADR(tyP0202OpsMag1.tyIOMonitor.tyBtnMag1FixedClampCtrl.uiRtStat));
	END_IF

	IF p_tyNtParamCurr.tyDOSettings.diMag1RemoteClampCtrl = 0 THEN
		fUIInRtStatHide(ADR(tyP0202OpsMag1.tyIOMonitor.tyBtnMag1RemoteClampCtrl.uiRtStat));
	END_IF

	IF p_tyNtParamCurr.tyDOSettings.diMag1ConvMtrIn = 0 THEN
		fUIInRtStatHide(ADR(tyP0202OpsMag1.tyIOMonitor.tyBtnMag1ConvMtrIn.uiRtStat));
	END_IF

	IF p_tyNtParamCurr.tyDOSettings.diMag1ConvMtrOut = 0 THEN
		fUIInRtStatHide(ADR(tyP0202OpsMag1.tyIOMonitor.tyBtnMag1ConvMtrOut.uiRtStat));
	END_IF

	tyP0202OpsMag1.tyIOMonitor.tyBtnMagSelClampCtrl.uiRtStat.0		:= NOT p_tyNtParamCurr.bMagAutoVerifyPrep;
	tyP0202OpsMag1.tyIOMonitor.tyBtnHeightSen.uiRtStat.0			:= NOT p_tyNtParamCurr.bMagAutoVerifyPrep;
	tyP0202OpsMag1.tyIOMonitor.tyBtnCAB717Sen.uiRtStat.0			:= NOT p_tyNtParamCurr.bMagAutoVerifyPrep;
	tyP0202OpsMag1.tyIOMonitor.tyBtnMagLargeSen.uiRtStat.0			:= NOT p_tyNtParamCurr.bMagAutoVerifyPrep;
	tyP0202OpsMag1.tyIOMonitor.tyBtnMagSmallSen.uiRtStat.0			:= NOT p_tyNtParamCurr.bMagAutoVerifyPrep;
	tyP0202OpsMag1.tyIOMonitor.tyBtnSelUnclampRS.uiRtStat.0			:= NOT p_tyNtParamCurr.bMagAutoVerifyPrep;
	tyP0202OpsMag1.tyIOMonitor.tyBtnMagSelUnClampCtrl.uiRtStat.0	:= NOT p_tyNtParamCurr.bMagAutoVerifyPrep;

	tyP0202OpsMag1.tyOps.tyBtnUnloadMag.uiRtStat.0 := NOT (p_tyNtParamCurr.bProjLifterMagPlatform AND NOT(p_tyNtParamCurr.bProjMagConvLane1Prep)) ;
	tyP0202OpsMag1.tyOps.tyBtnUnloadMag.uiMaskRtStat.0 := NOT (p_tyNtParamCurr.bProjLifterMagPlatform AND NOT(p_tyNtParamCurr.bProjMagConvLane1Prep)) ;
	tyP0202OpsMag1.tyOps.tyBitmapUnloadMag.uiRtStat.0 := NOT (p_tyNtParamCurr.bProjLifterMagPlatform AND NOT(p_tyNtParamCurr.bProjMagConvLane1Prep));
	tyP0202OpsMag1.tyOps.tyBtnChgMag.uiRtStat.0 := p_tyNtParamCurr.bProjLifterMagPlatform;

	tyP0202OpsMag1.tyIOMonitor.tyBtnCurtainSen.uiRtStat.0			:= NOT p_tyNtParamCurr.bCurtainSenPrep;
	tyP0202OpsMag1.tyIOMonitor.tyBtnCurtainSenPB.uiRtStat.0			:= NOT p_tyNtParamCurr.bCurtainSenPrep;
	tyP0202OpsMag1.tyIOMonitor.tyBtnCurtainSenPBLED.uiRtStat.0		:= NOT p_tyNtParamCurr.bCurtainSenPrep;
	tyP0202OpsMag1.tyIOMonitor.tyBtnMag1DetSen.uiRtStat.0			:= NOT p_tyNtParamCurr.bProjFixClprMagDetectSenPrep;

	tyP0202OpsMag1.tyChgMag.tyLyr.uiRtStat := NOT(p_tyNtParamCurr.bProjMagConvLane1Prep);
	IF p_tyNtParamCurr.eCustomerReq = Siemens THEN //Siemen
		tyP0202OpsMag1.tyIOMonitor.tyBtnTLAmber.usiTxtIdx := 25;
	END_IF

END_ACTION
```

#### Act_Main_P0203.st
```iecst
(** 2018-12-21 **)
ACTION Act_Main_P0203:

	//Machine Bitmap
	IF p_tyNtParamCurr.eProjMag = ULMagTriple THEN
		IF p_tyNtParamCurr.bProjLifterMagPlatform AND p_tyNtParamCurr.bUIConvDirRL THEN
			tyP0203OpsMag2.tyOps.tyBitmapMc.uiValueIdx	:= 800;
		ELSIF p_tyNtParamCurr.bProjLifterMagPlatform THEN
			tyP0203OpsMag2.tyOps.tyBitmapMc.uiValueIdx	:= 500;
		ELSE
			tyP0203OpsMag2.tyOps.tyBitmapMc.uiValueIdx	:= 200;
		END_IF

	ELSIF p_tyNtParamCurr.eProjMag = ULMagDual THEN
		IF p_tyNtParamCurr.bProjLifterMagPlatform AND p_tyNtParamCurr.bUIConvDirRL THEN
			tyP0203OpsMag2.tyOps.tyBitmapMc.uiValueIdx	:= 700;
		ELSIF p_tyNtParamCurr.bProjLifterMagPlatform AND p_tyNtParamCurr.bUIConvDirRL = FALSE AND p_tyNtParamCurr.bProjMagConvLane1Prep THEN
			tyP0203OpsMag2.tyOps.tyBitmapMc.uiValueIdx	:= 900;
		ELSIF p_tyNtParamCurr.bProjLifterMagPlatform THEN
			tyP0203OpsMag2.tyOps.tyBitmapMc.uiValueIdx	:= 600;
		ELSE
			tyP0203OpsMag2.tyOps.tyBitmapMc.uiValueIdx	:= 300;
		END_IF
	END_IF

	//AIV
//	tyP0203OpsMag2.tyOps.tyTxtLblAIV.uiRtStat.0		:= NOT p_tyNtParamCurr.bProjAGVPrep;
//	tyP0203OpsMag2.tyOps.tyBtnAIVWifi.uiRtStat.0	:= NOT p_tyNtParamCurr.bProjAGVPrep;
	tyP0203OpsMag2.tyOps.tyTxtLblAIV.uiRtStat.0		:= TRUE;
	tyP0203OpsMag2.tyOps.tyBtnAIVWifi.uiRtStat.0	:= TRUE;
	tyP0203OpsMag2.tyOps.tyBtnChgMag.uiRtStat.0		:= NOT(p_tyNtParamCurr.bProjAGVPrep AND p_tyNtParamCurr.bProjBtnInsertRmvMag);
	tyP0203OpsMag2.tyOps.tyBitmapChgMag.uiRtStat.0	:= NOT(p_tyNtParamCurr.bProjAGVPrep AND p_tyNtParamCurr.bProjBtnInsertRmvMag);

	//Display
	IF p_tyNtParamCurr.bProjLaneBPrep = FALSE THEN
		fUIInRtStatHide(ADR(tyP0203OpsMag2.tyIOMonitor.tyBtnUBAB.uiRtStat));
		fUIInRtStatHide(ADR(tyP0203OpsMag2.tyIOMonitor.tyBtnUBABStat.uiRtStat));
		fUIInRtStatHide(ADR(tyP0203OpsMag2.tyIOMonitor.tyBtnOvenInfeedSigB.uiRtStat));

		fUIInRtStatHide(ADR(tyP0203OpsMag2.tyIOMonitor.tyBtnUSBB.uiRtStat));
		fUIInRtStatHide(ADR(tyP0203OpsMag2.tyIOMonitor.tyBtnOvenInfoSigB.uiRtStat));
	END_IF

	IF p_tyNtParamCurr.bOvenInfoExtdPrep = FALSE THEN
		fUIInRtStatHide(ADR(tyP0203OpsMag2.tyIOMonitor.tyBtnOvenInfeedSigA.uiRtStat));
		fUIInRtStatHide(ADR(tyP0203OpsMag2.tyIOMonitor.tyBtnOvenInfeedSigB.uiRtStat));
	END_IF

	//Change Parameter
	IF p_tyNtParamCurr.bProjLaneBPrep THEN
		tyP0203OpsMag2.tyParam.tyDrpDnMcMode.usiValueMaxIdx	:= 8;
	ELSE
		tyP0203OpsMag2.tyParam.tyDrpDnMcMode.usiValueMaxIdx	:= 2;
	END_IF

	//Digital Input Used
	IF p_tyNtParamCurr.tyDISettings.diSafetyRlySig = 0 THEN
		fUIInRtStatHide(ADR(tyP0203OpsMag2.tyIOMonitor.tyBtnSafetyRlySig.uiRtStat));
	END_IF

	IF p_tyNtParamCurr.tyDISettings.diEStopSig = 0 THEN
		fUIInRtStatHide(ADR(tyP0203OpsMag2.tyIOMonitor.tyBtnEStop.uiRtStat));
	END_IF

	IF p_tyNtParamCurr.tyDISettings.diCoverSWSig = 0 THEN
		fUIInRtStatHide(ADR(tyP0203OpsMag2.tyIOMonitor.tyBtnCoverSWSig.uiRtStat));
	END_IF
	IF p_tyNtParamCurr.tyDISettings.diUBAA = 0 THEN
		fUIInRtStatHide(ADR(tyP0203OpsMag2.tyIOMonitor.tyBtnUBAA.uiRtStat));
	END_IF

	IF p_tyNtParamCurr.tyDISettings.diUBAAStat = 0 THEN
		fUIInRtStatHide(ADR(tyP0203OpsMag2.tyIOMonitor.tyBtnUBAAStat.uiRtStat));
	END_IF

	IF p_tyNtParamCurr.tyDISettings.diUBAB = 0 THEN
		fUIInRtStatHide(ADR(tyP0203OpsMag2.tyIOMonitor.tyBtnUBAB.uiRtStat));
	END_IF

	IF p_tyNtParamCurr.tyDISettings.diUBABStat = 0 THEN
		fUIInRtStatHide(ADR(tyP0203OpsMag2.tyIOMonitor.tyBtnUBABStat.uiRtStat));
	END_IF

	IF p_tyNtParamCurr.tyDISettings.diOvenInfeedSigA = 0 THEN
		fUIInRtStatHide(ADR(tyP0203OpsMag2.tyIOMonitor.tyBtnOvenInfeedSigA.uiRtStat));
	END_IF

	IF p_tyNtParamCurr.tyDISettings.diOvenInfeedSigB = 0 THEN
		fUIInRtStatHide(ADR(tyP0203OpsMag2.tyIOMonitor.tyBtnOvenInfeedSigB.uiRtStat));
	END_IF

	IF p_tyNtParamCurr.tyDISettings.diMag2FixedClampRS = 0 THEN
		fUIInRtStatHide(ADR(tyP0203OpsMag2.tyIOMonitor.tyBtnMag2FixedClmpRS.uiRtStat));
	END_IF

	IF p_tyNtParamCurr.tyDISettings.diMag2FixedUnclampRS = 0 THEN
		fUIInRtStatHide(ADR(tyP0203OpsMag2.tyIOMonitor.tyBtnMag2FixedUnclmpRS.uiRtStat));
	END_IF

	IF p_tyNtParamCurr.tyDISettings.diMag2RemoteClampRS = 0 THEN
		fUIInRtStatHide(ADR(tyP0203OpsMag2.tyIOMonitor.tyBtnMag2RmtClmpRS.uiRtStat));
	END_IF

	IF p_tyNtParamCurr.tyDISettings.diMag2RemoteUnclampRS = 0 THEN
		fUIInRtStatHide(ADR(tyP0203OpsMag2.tyIOMonitor.tyBtnMag2RmtUnclmpRS.uiRtStat));
	END_IF

	IF p_tyNtParamCurr.tyDISettings.diMagConvEntSen2 = 0 THEN
		fUIInRtStatHide(ADR(tyP0203OpsMag2.tyIOMonitor.tyBtnMag2ConvEntrySen.uiRtStat));
	END_IF

	IF p_tyNtParamCurr.tyDISettings.diMagPresentSen2 = 0 THEN
		fUIInRtStatHide(ADR(tyP0203OpsMag2.tyIOMonitor.tyBtnMag2PresentSen.uiRtStat));
	END_IF

	IF p_tyNtParamCurr.tyDISettings.diMag2AIVInPosSen1 = 0 THEN
		fUIInRtStatHide(ADR(tyP0203OpsMag2.tyIOMonitor.tyBtnMag2AIVInPosSen1.uiRtStat));
	END_IF

	IF p_tyNtParamCurr.tyDISettings.diMag2AIVInPosSen2 = 0 THEN
		fUIInRtStatHide(ADR(tyP0203OpsMag2.tyIOMonitor.tyBtnMag2AIVInPosSen2.uiRtStat));
	END_IF

	IF p_tyNtParamCurr.tyDISettings.diMag1OrientChkSen1 = 0 THEN
		fUIInRtStatHide(ADR(tyP0203OpsMag2.tyIOMonitor.tyBtnMag2OrientationChkSen1.uiRtStat));
	END_IF

	IF p_tyNtParamCurr.tyDISettings.diMag2OrientChkSen2 = 0 THEN
		fUIInRtStatHide(ADR(tyP0203OpsMag2.tyIOMonitor.tyBtnMag2OrientationChkSen2.uiRtStat));
	END_IF

	//Digital Output Selected
	IF p_tyNtParamCurr.tyDOSettings.diSafetyRlyRst = 0 THEN
		fUIInRtStatHide(ADR(tyP0203OpsMag2.tyIOMonitor.tyBtnSafetyRlyRst.uiRtStat));
	END_IF

	IF p_tyNtParamCurr.tyDOSettings.diTLGreen = 0 THEN
		fUIInRtStatHide(ADR(tyP0203OpsMag2.tyIOMonitor.tyBtnTLGreen.uiRtStat));
	END_IF

	IF p_tyNtParamCurr.tyDOSettings.diTLAmber = 0 THEN
		fUIInRtStatHide(ADR(tyP0203OpsMag2.tyIOMonitor.tyBtnTLAmber.uiRtStat));
	END_IF

	IF p_tyNtParamCurr.tyDOSettings.diTLRed = 0 THEN
		fUIInRtStatHide(ADR(tyP0203OpsMag2.tyIOMonitor.tyBtnTLRed.uiRtStat));
	END_IF

	IF p_tyNtParamCurr.tyDOSettings.diBuzzer = 0 THEN
		fUIInRtStatHide(ADR(tyP0203OpsMag2.tyIOMonitor.tyBtnBuzzer.uiRtStat));
	END_IF

	IF p_tyNtParamCurr.tyDOSettings.diUSBA = 0 THEN
		fUIInRtStatHide(ADR(tyP0203OpsMag2.tyIOMonitor.tyBtnUSBA.uiRtStat));
	END_IF

	IF p_tyNtParamCurr.tyDOSettings.diUSBB = 0 THEN
		fUIInRtStatHide(ADR(tyP0203OpsMag2.tyIOMonitor.tyBtnUSBB.uiRtStat));
	END_IF

	IF p_tyNtParamCurr.tyDOSettings.diOvenInfoSigA = 0 THEN
		fUIInRtStatHide(ADR(tyP0203OpsMag2.tyIOMonitor.tyBtnOvenInfoSigA.uiRtStat));
	END_IF

	IF p_tyNtParamCurr.tyDOSettings.diOvenInfoSigB = 0 THEN
		fUIInRtStatHide(ADR(tyP0203OpsMag2.tyIOMonitor.tyBtnOvenInfoSigB.uiRtStat));
	END_IF

	IF p_tyNtParamCurr.tyDOSettings.diMag2FixedClampCtrl = 0 THEN
		fUIInRtStatHide(ADR(tyP0203OpsMag2.tyIOMonitor.tyBtnMag2FixedClampCtrl.uiRtStat));
	END_IF

	IF p_tyNtParamCurr.tyDOSettings.diMag2RemoteClampCtrl = 0 THEN
		fUIInRtStatHide(ADR(tyP0203OpsMag2.tyIOMonitor.tyBtnMag2RemoteClampCtrl.uiRtStat));
	END_IF

	IF p_tyNtParamCurr.tyDOSettings.diMag2ConvMtrIn = 0 THEN
		fUIInRtStatHide(ADR(tyP0203OpsMag2.tyIOMonitor.tyBtnMag2ConvMtrIn.uiRtStat));
	END_IF

	IF p_tyNtParamCurr.tyDOSettings.diMag2ConvMtrOut = 0 THEN
		fUIInRtStatHide(ADR(tyP0203OpsMag2.tyIOMonitor.tyBtnMag2ConvMtrOut.uiRtStat));
	END_IF

	tyP0203OpsMag2.tyIOMonitor.tyBtnMagSelClampCtrl.uiRtStat.0		:= NOT p_tyNtParamCurr.bMagAutoVerifyPrep;
	tyP0203OpsMag2.tyIOMonitor.tyBtnHeightSen.uiRtStat.0			:= NOT p_tyNtParamCurr.bMagAutoVerifyPrep;
	tyP0203OpsMag2.tyIOMonitor.tyBtnCAB717Sen.uiRtStat.0			:= NOT p_tyNtParamCurr.bMagAutoVerifyPrep;
	tyP0203OpsMag2.tyIOMonitor.tyBtnMagLargeSen.uiRtStat.0			:= NOT p_tyNtParamCurr.bMagAutoVerifyPrep;
	tyP0203OpsMag2.tyIOMonitor.tyBtnMagSmallSen.uiRtStat.0			:= NOT p_tyNtParamCurr.bMagAutoVerifyPrep;
	tyP0203OpsMag2.tyIOMonitor.tyBtnSelUnclampRS.uiRtStat.0			:= NOT p_tyNtParamCurr.bMagAutoVerifyPrep;
	tyP0203OpsMag2.tyIOMonitor.tyBtnMagSelUnClampCtrl.uiRtStat.0	:= NOT p_tyNtParamCurr.bMagAutoVerifyPrep;

	IF p_tyNtParamCurr.eProjMag = ULMagTriple AND p_tyNtParamCurr.bMagAutoVerifyPrep = TRUE THEN
		tyP0203OpsMag2.tyOps.tyBitmapMc.usiValueIdx	:= 200;
	ELSE
		tyP0203OpsMag2.tyOps.tyBitmapMc.usiValueIdx	:= 0;
	END_IF

	tyP0203OpsMag2.tyOps.tyBtnUnloadMag.uiRtStat.0 := NOT (p_tyNtParamCurr.bProjLifterMagPlatform AND NOT(p_tyNtParamCurr.bProjMagConvLane2Prep));
	tyP0203OpsMag2.tyOps.tyBtnUnloadMag.uiMaskRtStat.0 := NOT (p_tyNtParamCurr.bProjLifterMagPlatform AND NOT(p_tyNtParamCurr.bProjMagConvLane2Prep)) ;
	tyP0203OpsMag2.tyOps.tyBitmapUnloadMag.uiRtStat.0 := NOT (p_tyNtParamCurr.bProjLifterMagPlatform AND NOT(p_tyNtParamCurr.bProjMagConvLane2Prep));
	tyP0203OpsMag2.tyOps.tyBtnChgMag.uiRtStat.0 := p_tyNtParamCurr.bProjLifterMagPlatform;

	tyP0203OpsMag2.tyIOMonitor.tyBtnCurtainSen.uiRtStat.0			:= NOT p_tyNtParamCurr.bCurtainSenPrep;
	tyP0203OpsMag2.tyIOMonitor.tyBtnCurtainSenPB.uiRtStat.0			:= NOT p_tyNtParamCurr.bCurtainSenPrep;
	tyP0203OpsMag2.tyIOMonitor.tyBtnCurtainSenPBLED.uiRtStat.0		:= NOT p_tyNtParamCurr.bCurtainSenPrep;

	tyP0203OpsMag2.tyIOMonitor.tyBtnMag2DetSen.uiRtStat.0			:= NOT p_tyNtParamCurr.bProjFixClprMagDetectSenPrep;

	tyP0203OpsMag2.tyChgMag.tyLyr.uiRtStat := NOT(p_tyNtParamCurr.bProjMagConvLane2Prep);
	IF p_tyNtParamCurr.eCustomerReq = Siemens THEN //Siemen
		tyP0203OpsMag2.tyIOMonitor.tyBtnTLAmber.usiTxtIdx := 25;
	END_IF

END_ACTION
```

#### Act_Main_P0204.st
```iecst
(** 2018-12-21 **)
ACTION Act_Main_P0204:

	//Machine Bitmap
	IF p_tyNtParamCurr.eProjMag = ULMagTriple THEN
		IF p_tyNtParamCurr.bProjLifterMagPlatform AND p_tyNtParamCurr.bUIConvDirRL THEN
			tyP0204OpsMag3.tyOps.tyBitmapMc.uiValueIdx	:= 800;
		ELSIF p_tyNtParamCurr.bProjLifterMagPlatform THEN
			tyP0204OpsMag3.tyOps.tyBitmapMc.uiValueIdx	:= 500;
		ELSE
			tyP0204OpsMag3.tyOps.tyBitmapMc.uiValueIdx	:= 200;
		END_IF
	ELSIF p_tyNtParamCurr.eProjMag = ULMagDual THEN
		IF p_tyNtParamCurr.bProjLifterMagPlatform AND p_tyNtParamCurr.bUIConvDirRL THEN
			tyP0204OpsMag3.tyOps.tyBitmapMc.uiValueIdx	:= 700;
		ELSIF p_tyNtParamCurr.bProjLifterMagPlatform THEN
			tyP0204OpsMag3.tyOps.tyBitmapMc.uiValueIdx	:= 600;
		ELSE
			tyP0204OpsMag3.tyOps.tyBitmapMc.uiValueIdx	:= 0;
		END_IF
	END_IF

	//AIV
//	tyP0204OpsMag3.tyOps.tyTxtLblAIV.uiRtStat.0		:= NOT p_tyNtParamCurr.bProjAGVPrep;
//	tyP0204OpsMag3.tyOps.tyBtnAIVWifi.uiRtStat.0	:= NOT p_tyNtParamCurr.bProjAGVPrep;
	tyP0204OpsMag3.tyOps.tyTxtLblAIV.uiRtStat.0		:= TRUE;
	tyP0204OpsMag3.tyOps.tyBtnAIVWifi.uiRtStat.0	:= TRUE;
	tyP0204OpsMag3.tyOps.tyBtnChgMag.uiRtStat.0		:= NOT(p_tyNtParamCurr.bProjAGVPrep AND p_tyNtParamCurr.bProjBtnInsertRmvMag);
	tyP0204OpsMag3.tyOps.tyBitmapChgMag.uiRtStat.0	:= NOT(p_tyNtParamCurr.bProjAGVPrep AND p_tyNtParamCurr.bProjBtnInsertRmvMag);

	//Display
	IF p_tyNtParamCurr.bProjLaneBPrep = FALSE THEN
		fUIInRtStatHide(ADR(tyP0204OpsMag3.tyIOMonitor.tyBtnUBAB.uiRtStat));
		fUIInRtStatHide(ADR(tyP0204OpsMag3.tyIOMonitor.tyBtnUBABStat.uiRtStat));
		fUIInRtStatHide(ADR(tyP0204OpsMag3.tyIOMonitor.tyBtnOvenInfeedSigB.uiRtStat));

		fUIInRtStatHide(ADR(tyP0204OpsMag3.tyIOMonitor.tyBtnUSBB.uiRtStat));
		fUIInRtStatHide(ADR(tyP0204OpsMag3.tyIOMonitor.tyBtnOvenInfoSigB.uiRtStat));
	END_IF

	IF p_tyNtParamCurr.bOvenInfoExtdPrep = FALSE THEN
		fUIInRtStatHide(ADR(tyP0204OpsMag3.tyIOMonitor.tyBtnOvenInfeedSigA.uiRtStat));
		fUIInRtStatHide(ADR(tyP0204OpsMag3.tyIOMonitor.tyBtnOvenInfeedSigB.uiRtStat));
	END_IF

	//Change Parameter
	IF p_tyNtParamCurr.bProjLaneBPrep THEN
		tyP0204OpsMag3.tyParam.tyDrpDnMcMode.usiValueMaxIdx	:= 8;
	ELSE
		tyP0204OpsMag3.tyParam.tyDrpDnMcMode.usiValueMaxIdx	:= 2;
	END_IF

	//Digital Input Used
	IF p_tyNtParamCurr.tyDISettings.diSafetyRlySig = 0 THEN
		fUIInRtStatHide(ADR(tyP0204OpsMag3.tyIOMonitor.tyBtnSafetyRlySig.uiRtStat));
	END_IF

	IF p_tyNtParamCurr.tyDISettings.diEStopSig = 0 THEN
		fUIInRtStatHide(ADR(tyP0204OpsMag3.tyIOMonitor.tyBtnEStop.uiRtStat));
	END_IF

	IF p_tyNtParamCurr.tyDISettings.diCoverSWSig = 0 THEN
		fUIInRtStatHide(ADR(tyP0204OpsMag3.tyIOMonitor.tyBtnCoverSWSig.uiRtStat));
	END_IF

	IF p_tyNtParamCurr.tyDISettings.diUBAA = 0 THEN
		fUIInRtStatHide(ADR(tyP0204OpsMag3.tyIOMonitor.tyBtnUBAA.uiRtStat));
	END_IF

	IF p_tyNtParamCurr.tyDISettings.diUBAAStat = 0 THEN
		fUIInRtStatHide(ADR(tyP0204OpsMag3.tyIOMonitor.tyBtnUBAAStat.uiRtStat));
	END_IF

	IF p_tyNtParamCurr.tyDISettings.diUBAB = 0 THEN
		fUIInRtStatHide(ADR(tyP0204OpsMag3.tyIOMonitor.tyBtnUBAB.uiRtStat));
	END_IF

	IF p_tyNtParamCurr.tyDISettings.diUBABStat = 0 THEN
		fUIInRtStatHide(ADR(tyP0204OpsMag3.tyIOMonitor.tyBtnUBABStat.uiRtStat));
	END_IF

	IF p_tyNtParamCurr.tyDISettings.diOvenInfeedSigA = 0 THEN
		fUIInRtStatHide(ADR(tyP0204OpsMag3.tyIOMonitor.tyBtnOvenInfeedSigA.uiRtStat));
	END_IF

	IF p_tyNtParamCurr.tyDISettings.diOvenInfeedSigB = 0 THEN
		fUIInRtStatHide(ADR(tyP0204OpsMag3.tyIOMonitor.tyBtnOvenInfeedSigB.uiRtStat));
	END_IF

	IF p_tyNtParamCurr.tyDISettings.diMag3FixedClampRS = 0 THEN
		fUIInRtStatHide(ADR(tyP0204OpsMag3.tyIOMonitor.tyBtnMag3FixedClmpRS.uiRtStat));
	END_IF

	IF p_tyNtParamCurr.tyDISettings.diMag3FixedUnclampRS = 0 THEN
		fUIInRtStatHide(ADR(tyP0204OpsMag3.tyIOMonitor.tyBtnMag3FixedUnclmpRS.uiRtStat));
	END_IF

	IF p_tyNtParamCurr.tyDISettings.diMag3RemoteClampRS = 0 THEN
		fUIInRtStatHide(ADR(tyP0204OpsMag3.tyIOMonitor.tyBtnMag3RmtClmpRS.uiRtStat));
	END_IF

	IF p_tyNtParamCurr.tyDISettings.diMag3RemoteUnclampRS = 0 THEN
		fUIInRtStatHide(ADR(tyP0204OpsMag3.tyIOMonitor.tyBtnMag3RmtUnclmpRS.uiRtStat));
	END_IF

	IF p_tyNtParamCurr.tyDISettings.diMagConvEntSen3 = 0 THEN
		fUIInRtStatHide(ADR(tyP0204OpsMag3.tyIOMonitor.tyBtnMag3ConvEntrySen.uiRtStat));
	END_IF

	IF p_tyNtParamCurr.tyDISettings.diMagPresentSen3 = 0 THEN
		fUIInRtStatHide(ADR(tyP0204OpsMag3.tyIOMonitor.tyBtnMag3PresentSen.uiRtStat));
	END_IF

	IF p_tyNtParamCurr.tyDISettings.diMag3AIVInPosSen1 = 0 THEN
		fUIInRtStatHide(ADR(tyP0204OpsMag3.tyIOMonitor.tyBtnMag3AIVInPosSen1.uiRtStat));
	END_IF

	IF p_tyNtParamCurr.tyDISettings.diMag3AIVInPosSen2 = 0 THEN
		fUIInRtStatHide(ADR(tyP0204OpsMag3.tyIOMonitor.tyBtnMag3AIVInPosSen2.uiRtStat));
	END_IF

	IF p_tyNtParamCurr.tyDISettings.diMag3OrientChkSen1 = 0 THEN
		fUIInRtStatHide(ADR(tyP0204OpsMag3.tyIOMonitor.tyBtnMag3OrientationChkSen1.uiRtStat));
	END_IF

	IF p_tyNtParamCurr.tyDISettings.diMag3OrientChkSen2 = 0 THEN
		fUIInRtStatHide(ADR(tyP0204OpsMag3.tyIOMonitor.tyBtnMag3OrientationChkSen2.uiRtStat));
	END_IF

	//Digital Output Selected
	IF p_tyNtParamCurr.tyDOSettings.diSafetyRlyRst = 0 THEN
		fUIInRtStatHide(ADR(tyP0204OpsMag3.tyIOMonitor.tyBtnSafetyRlyRst.uiRtStat));
	END_IF

	IF p_tyNtParamCurr.tyDOSettings.diTLGreen = 0 THEN
		fUIInRtStatHide(ADR(tyP0204OpsMag3.tyIOMonitor.tyBtnTLGreen.uiRtStat));
	END_IF

	IF p_tyNtParamCurr.tyDOSettings.diTLAmber = 0 THEN
		fUIInRtStatHide(ADR(tyP0204OpsMag3.tyIOMonitor.tyBtnTLAmber.uiRtStat));
	END_IF

	IF p_tyNtParamCurr.tyDOSettings.diTLRed = 0 THEN
		fUIInRtStatHide(ADR(tyP0204OpsMag3.tyIOMonitor.tyBtnTLRed.uiRtStat));
	END_IF

	IF p_tyNtParamCurr.tyDOSettings.diBuzzer = 0 THEN
		fUIInRtStatHide(ADR(tyP0204OpsMag3.tyIOMonitor.tyBtnBuzzer.uiRtStat));
	END_IF

	IF p_tyNtParamCurr.tyDOSettings.diUSBA = 0 THEN
		fUIInRtStatHide(ADR(tyP0204OpsMag3.tyIOMonitor.tyBtnUSBA.uiRtStat));
	END_IF

	IF p_tyNtParamCurr.tyDOSettings.diUSBB = 0 THEN
		fUIInRtStatHide(ADR(tyP0204OpsMag3.tyIOMonitor.tyBtnUSBB.uiRtStat));
	END_IF

	IF p_tyNtParamCurr.tyDOSettings.diOvenInfoSigA = 0 THEN
		fUIInRtStatHide(ADR(tyP0204OpsMag3.tyIOMonitor.tyBtnOvenInfoSigA.uiRtStat));
	END_IF

	IF p_tyNtParamCurr.tyDOSettings.diOvenInfoSigB = 0 THEN
		fUIInRtStatHide(ADR(tyP0204OpsMag3.tyIOMonitor.tyBtnOvenInfoSigB.uiRtStat));
	END_IF

	IF p_tyNtParamCurr.tyDOSettings.diMag3FixedClampCtrl = 0 THEN
		fUIInRtStatHide(ADR(tyP0204OpsMag3.tyIOMonitor.tyBtnMag3FixedClampCtrl.uiRtStat));
	END_IF

	IF p_tyNtParamCurr.tyDOSettings.diMag3RemoteClampCtrl = 0 THEN
		fUIInRtStatHide(ADR(tyP0204OpsMag3.tyIOMonitor.tyBtnMag3RemoteClampCtrl.uiRtStat));
	END_IF

	IF p_tyNtParamCurr.tyDOSettings.diMag3ConvMtrIn = 0 THEN
		fUIInRtStatHide(ADR(tyP0204OpsMag3.tyIOMonitor.tyBtnMag3ConvMtrIn.uiRtStat));
	END_IF

	IF p_tyNtParamCurr.tyDOSettings.diMag3ConvMtrOut = 0 THEN
		fUIInRtStatHide(ADR(tyP0204OpsMag3.tyIOMonitor.tyBtnMag3ConvMtrOut.uiRtStat));
	END_IF

	tyP0204OpsMag3.tyIOMonitor.tyBtnMagSelClampCtrl.uiRtStat.0		:= NOT p_tyNtParamCurr.bMagAutoVerifyPrep;
	tyP0204OpsMag3.tyIOMonitor.tyBtnHeightSen.uiRtStat.0			:= NOT p_tyNtParamCurr.bMagAutoVerifyPrep;
	tyP0204OpsMag3.tyIOMonitor.tyBtnCAB717Sen.uiRtStat.0			:= NOT p_tyNtParamCurr.bMagAutoVerifyPrep;
	tyP0204OpsMag3.tyIOMonitor.tyBtnMagLargeSen.uiRtStat.0			:= NOT p_tyNtParamCurr.bMagAutoVerifyPrep;
	tyP0204OpsMag3.tyIOMonitor.tyBtnMagSmallSen.uiRtStat.0			:= NOT p_tyNtParamCurr.bMagAutoVerifyPrep;
	tyP0204OpsMag3.tyIOMonitor.tyBtnSelUnclampRS.uiRtStat.0			:= NOT p_tyNtParamCurr.bMagAutoVerifyPrep;
	tyP0204OpsMag3.tyIOMonitor.tyBtnMagSelUnClampCtrl.uiRtStat.0	:= NOT p_tyNtParamCurr.bMagAutoVerifyPrep;

	tyP0204OpsMag3.tyOps.tyBtnUnloadMag.uiRtStat.0 := NOT p_tyNtParamCurr.bProjLifterMagPlatform;
	tyP0204OpsMag3.tyOps.tyBtnUnloadMag.uiMaskRtStat.0 := NOT p_tyNtParamCurr.bProjLifterMagPlatform  ;
	tyP0204OpsMag3.tyOps.tyBitmapUnloadMag.uiRtStat.0 := NOT p_tyNtParamCurr.bProjLifterMagPlatform;
	tyP0204OpsMag3.tyOps.tyBtnChgMag.uiRtStat.0 := p_tyNtParamCurr.bProjLifterMagPlatform;

	tyP0204OpsMag3.tyIOMonitor.tyBtnCurtainSen.uiRtStat.0			:= NOT p_tyNtParamCurr.bCurtainSenPrep;
	tyP0204OpsMag3.tyIOMonitor.tyBtnCurtainSenPB.uiRtStat.0			:= NOT p_tyNtParamCurr.bCurtainSenPrep;
	tyP0204OpsMag3.tyIOMonitor.tyBtnCurtainSenPBLED.uiRtStat.0		:= NOT p_tyNtParamCurr.bCurtainSenPrep;

	tyP0204OpsMag3.tyIOMonitor.tyBtnMag3DetSen.uiRtStat.0			:= NOT p_tyNtParamCurr.bProjFixClprMagDetectSenPrep;

	IF p_tyNtParamCurr.eCustomerReq = Siemens THEN //Siemen
		tyP0204OpsMag3.tyIOMonitor.tyBtnTLAmber.usiTxtIdx := 25;
	END_IF
END_ACTION
```

#### Act_Main_P0205.st
```iecst
(** 2021-05-14 **)
ACTION Act_Main_P0205:

	//Machine Bitmap
	IF p_tyNtParamCurr.eProjMag = ULMagDual THEN
		fUIInRtStatHide(ADR(tyP0205OpsAIV.tyIOMonitor.tyTripleMagLyr.uiRtStat));
		fUIInRtStatOff(ADR(tyP0205OpsAIV.tyIOMonitor.tyDualMagLyr.uiRtStat));
	ELSIF p_tyNtParamCurr.eProjMag = ULMagTriple THEN
		fUIInRtStatHide(ADR(tyP0205OpsAIV.tyIOMonitor.tyDualMagLyr.uiRtStat));
		fUIInRtStatOff(ADR(tyP0205OpsAIV.tyIOMonitor.tyTripleMagLyr.uiRtStat));
	END_IF

	tyP0205OpsAIV.tyIOMonitor.tyBtnAIVSotRCVOk1.uiRtStat.0 := NOT(p_tyNtParamCurr.bProjSOTSensorPrep);
	tyP0205OpsAIV.tyIOMonitor.tyBtnAIVSotRCVOk2.uiRtStat.0 := NOT(p_tyNtParamCurr.bProjSOTSensorPrep);
	tyP0205OpsAIV.tyIOMonitor.tyBtnAIVSotRCVOk3.uiRtStat.0 := NOT(p_tyNtParamCurr.bProjSOTSensorPrep);
	tyP0205OpsAIV.tyIOMonitor.tyBtnAIVSotRCVOk4.uiRtStat.0 := NOT(p_tyNtParamCurr.bProjSOTSensorPrep);

	tyP0205OpsAIV.tyIOMonitor.tyStringMesName.uiRtStat.0 := NOT(p_tyNtParamCurr.bShowMESName);
	IF p_tyNtParamCurr.bShowFMorMESActive THEN
		tyP0205OpsAIV.tyIOMonitor.tyBtnMESActive.usiTxtIdx := 6;
	ELSE
		tyP0205OpsAIV.tyIOMonitor.tyBtnMESActive.usiTxtIdx := 0;
	END_IF

	IF p_tyMcParamCurr.eAGVComProtocol =  McSetAGVTCPEnableTCP THEN
		tyP0205OpsAIV.tyIOMonitor.tyBtnMESActive.uiRtStat 		:= TRUE;
		tyP0205OpsAIV.tyIOMonitor.tyBtnReqAIVToBring1.uiRtStat 	:= TRUE;
		tyP0205OpsAIV.tyIOMonitor.tyBtnReqAIVToGet1.uiRtStat 	:= TRUE;
		tyP0205OpsAIV.tyIOMonitor.tyBtnReqAIVToBring2.uiRtStat 	:= TRUE;
		tyP0205OpsAIV.tyIOMonitor.tyBtnReqAIVToGet2.uiRtStat 	:= TRUE;

		tyP0205OpsAIV.tyIOMonitor.tyHotspotGroupError1.uiRtStat := TRUE;
		tyP0205OpsAIV.tyIOMonitor.tyHotspotGroupError2.uiRtStat := TRUE;
	END_IF

	//Siemens 3LD
	tyP0205OpsAIV.tyIOMonitor.tyBtnReqAIVToBring1.uiRtStat.0 := TRUE ; //p_tyNtParamCurr.eCustomerReq = Siemens;
	tyP0205OpsAIV.tyIOMonitor.tyBtnReqAIVToGet1.uiRtStat.0 := TRUE ; //p_tyNtParamCurr.eCustomerReq = Siemens;
	tyP0205OpsAIV.tyIOMonitor.tyBtnReqAIVToBring2.uiRtStat.0 := TRUE ; //p_tyNtParamCurr.eCustomerReq = Siemens;
	tyP0205OpsAIV.tyIOMonitor.tyBtnReqAIVToGet2.uiRtStat.0 := TRUE ; //p_tyNtParamCurr.eCustomerReq = Siemens;
	tyP0205OpsAIV.tyIOMonitor.tyBtnReqAIVToBring3.uiRtStat.0 := TRUE ; //p_tyNtParamCurr.eCustomerReq = Siemens;
	tyP0205OpsAIV.tyIOMonitor.tyBtnReqAIVToGet3.uiRtStat.0 := TRUE ; //p_tyNtParamCurr.eCustomerReq = Siemens;
END_ACTION
```

#### Act_Main_P0206.st
```iecst
(** 2021-05-14 **)
ACTION Act_Main_P0206:
	//Display
	IF p_tyNtParamCurr.bProjMagConvLane1Prep THEN
		tyP0206OpsMagConv1.tyIOMonitor.tyBtnEntStprExt.uiRtStat :=  NOT (p_bStopper1TwoCtrlOut);
		tyP0206OpsMagConv1.tyIOMonitor.tyBtnMidStprRet.uiRtStat :=  NOT (p_bStopper2TwoCtrlOut);
		tyP0206OpsMagConv1.tyIOMonitor.tyBtnExtStprExt.uiRtStat :=  NOT (p_bStopper3TwoCtrlOut);
		tyP0206OpsMagConv1.tyIOMonitor.tyBtnMidStprRet1.uiRtStat :=  NOT (p_bStopper4TwoCtrlOut);
		tyP0206OpsMagConv1.tyIOMonitor.tyBtnExtStprExt1.uiRtStat :=  NOT (p_bStopper5TwoCtrlOut);
	END_IF

END_ACTION
```

#### Act_Main_P0207.st
```iecst
(** 2021-05-14 **)
ACTION Act_Main_P0207:

	//Display
	IF p_tyNtParamCurr.bProjMagConvLane2Prep THEN
		tyP0207OpsMagConv2.tyIOMonitor.tyBtnEntStprExt.uiRtStat :=  NOT (p_bStopper1TwoCtrlOut2);
		tyP0207OpsMagConv2.tyIOMonitor.tyBtnMidStprRet.uiRtStat :=  NOT (p_bStopper2TwoCtrlOut2);
		tyP0207OpsMagConv2.tyIOMonitor.tyBtnExtStprExt.uiRtStat :=  NOT (p_bStopper3TwoCtrlOut2);
		tyP0207OpsMagConv2.tyIOMonitor.tyBtnMidStprRet1.uiRtStat :=  NOT (p_bStopper4TwoCtrlOut2);
		tyP0207OpsMagConv2.tyIOMonitor.tyBtnExtStprExt1.uiRtStat :=  NOT (p_bStopper5TwoCtrlOut2);
	END_IF

END_ACTION
```

#### Act_Main_P0400.st
```iecst
ACTION Act_Main_P0400:

	//Board Per Slot
	tyP0400ProdSel.tyProdSel.tyNumBrdPerSlt.uiRtStat.0		:= NOT p_tyNtParamCurr.bProjBrdPerSltPrep;
	tyP0400ProdSel.tyProdSel.tyTxtBrdPerSlt.uiRtStat.0		:= NOT p_tyNtParamCurr.bProjBrdPerSltPrep;
	tyP0400ProdSel.tyRcpDet.tyNumBrdPerSlt.uiRtStat.0		:= NOT p_tyNtParamCurr.bProjBrdPerSltPrep;
	tyP0400ProdSel.tyRcpDet.tyTxtBrdPerSlt.uiRtStat.0		:= NOT p_tyNtParamCurr.bProjBrdPerSltPrep;

	//Min Req To Free Buffer
	tyP0400ProdSel.tyProdSel.tyNumMinReqFreeBffr.uiRtStat.0	:= NOT p_tyNtParamCurr.bOvenInfoPrep;
	tyP0400ProdSel.tyProdSel.tyTxtMinReqFreeBffr.uiRtStat.0	:= NOT p_tyNtParamCurr.bOvenInfoPrep;
	tyP0400ProdSel.tyRcpDet.tyNumMinReqFreeBffr.uiRtStat.0	:= NOT p_tyNtParamCurr.bOvenInfoPrep;
	tyP0400ProdSel.tyRcpDet.tyTxtMinReqFreeBffr.uiRtStat.0	:= NOT p_tyNtParamCurr.bOvenInfoPrep;

	//Product Selection
	tyP0400ProdSel.tyProdSel.tyStringRecipeNm.sValue		:= p_tyProdRcpCurrRcp0.sRcpNm;
	tyP0400ProdSel.tyProdSel.tyNumProdWidth.diValue			:= p_tyProdRcpCurrRcp0.diWidthInUM;
	tyP0400ProdSel.tyProdSel.tyNumMaxSlt.diValue			:= p_tyProdRcpCurrRcp0.diMaxSltValue;
	tyP0400ProdSel.tyProdSel.tyNumMinSlt.diValue			:= p_tyProdRcpCurrRcp0.diMinSltValue;
	tyP0400ProdSel.tyProdSel.tyNumPitch.diValue				:= p_tyProdRcpCurrRcp0.diPitch;
	tyP0400ProdSel.tyProdSel.tyNumBrdPerSlt.diValue			:= p_tyProdRcpCurrRcp0.diBrdPerSlt;
	tyP0400ProdSel.tyProdSel.tyBtnToptoBtm.bValue			:= p_tyProdRcpCurrRcp0.bTopToBtm;
	tyP0400ProdSel.tyProdSel.tyBtnGapBetBrds.bValue			:= p_tyProdRcpCurrRcp0.bGapBwtnBrd;
	tyP0400ProdSel.tyProdSel.tyBtnLongBrd.bValue			:= p_tyProdRcpCurrRcp0.bLongBrd;
	tyP0400ProdSel.tyProdSel.tyTxtMcMode.usiValueIdx		:= p_tyProdRcpCurrRcp0.usiMcMod;
	tyP0400ProdSel.tyProdSel.tyNumMinReqFreeBffr.diValue	:= p_tyProdRcpCurrRcp0.diMinReqFreeBffr;
	tyP0400ProdSel.tyProdSel.tyNumPshrOffset.diValue		:= p_tyProdRcpCurrRcp0.diPshrOffset;

	//Motorized Pusher
	tyP0400ProdSel.tyProdSel.tyTxtMtrPshrExtSpd.uiRtStat.0	:= NOT p_tyNtParamCurr.bProjMotorizedPusherPrep;
	tyP0400ProdSel.tyProdSel.tyTxtMtrPshrExtTorq.uiRtStat.0	:= NOT p_tyNtParamCurr.bProjMotorizedPusherPrep;
	tyP0400ProdSel.tyProdSel.tyNumMtrPshrExtSpd.uiRtStat.0	:= NOT p_tyNtParamCurr.bProjMotorizedPusherPrep;
	tyP0400ProdSel.tyProdSel.tyNumMtrPshrExtTorq.uiRtStat.0	:= NOT p_tyNtParamCurr.bProjMotorizedPusherPrep;
	tyP0400ProdSel.tyRcpDet.tyTxtMtrPshrExtSpd.uiRtStat.0	:= NOT p_tyNtParamCurr.bProjMotorizedPusherPrep;
	tyP0400ProdSel.tyRcpDet.tyTxtMtrPshrExtTorq.uiRtStat.0	:= NOT p_tyNtParamCurr.bProjMotorizedPusherPrep;
	tyP0400ProdSel.tyRcpDet.tyNumMtrPshrExtSpd.uiRtStat.0	:= NOT p_tyNtParamCurr.bProjMotorizedPusherPrep;
	tyP0400ProdSel.tyRcpDet.tyNumMtrPshrExtTorq.uiRtStat.0	:= NOT p_tyNtParamCurr.bProjMotorizedPusherPrep;
	tyP0400ProdSel.tyProdSel.tyNumMtrPshrExtSpd.diValue		:= p_tyProdRcpCurrRcp0.diMtrPshrExtSpd;
	tyP0400ProdSel.tyProdSel.tyNumMtrPshrExtTorq.diValue	:= p_tyProdRcpCurrRcp0.diMtrPshrExtTorq;

	//Puller Offset
	tyP0400ProdSel.tyProdSel.tyNumPshrOffset.uiRtStat.0		:= NOT p_tyNtParamCurr.bAWPusherPrep;
	tyP0400ProdSel.tyProdSel.tyTxtPshrOffset.uiRtStat.0		:= NOT p_tyNtParamCurr.bAWPusherPrep;
	tyP0400ProdSel.tyRcpDet.tyNumPshrOffset.uiRtStat.0		:= NOT p_tyNtParamCurr.bAWPusherPrep;
	tyP0400ProdSel.tyRcpDet.tyTxtPshrOffset.uiRtStat.0		:= NOT p_tyNtParamCurr.bAWPusherPrep;

END_ACTION
```

#### Act_Main_P0410.st
```iecst
ACTION Act_Main_P0410:

	//Display
	tyP0410MagSel.tyMagSel.tyTxtLifMag3Slt1PosLbl.uiRtStat.0	:= NOT(p_tyNtParamCurr.eProjMag = ULMagTriple);
	tyP0410MagSel.tyMagSel.tyNumLifterMag3Slt1Pos.uiRtStat.0	:= NOT(p_tyNtParamCurr.eProjMag = ULMagTriple);

	tyP0410MagSel.tyMagDet.tyTxtLifMag3Slt1PosLbl.uiRtStat.0	:= NOT(p_tyNtParamCurr.eProjMag = ULMagTriple);
	tyP0410MagSel.tyMagDet.tyNumLifterMag3Slt1Pos.uiRtStat.0	:= NOT(p_tyNtParamCurr.eProjMag = ULMagTriple);

	tyP0410MagSel.tyMagSel.tyTxtTravPosMag3Lbl.uiRtStat.0	:= NOT(p_tyNtParamCurr.eProjMag = ULMagTriple);
	tyP0410MagSel.tyMagSel.tyNumTravPosMag3.uiRtStat.0		:= NOT(p_tyNtParamCurr.eProjMag = ULMagTriple);

	tyP0410MagSel.tyMagDet.tyTxtTravPosMag3Lbl.uiRtStat.0	:= NOT(p_tyNtParamCurr.eProjMag = ULMagTriple);
	tyP0410MagSel.tyMagDet.tyNumTravPosMag3.uiRtStat.0		:= NOT(p_tyNtParamCurr.eProjMag = ULMagTriple);

	//Magazine Selection
	tyP0410MagSel.tyMagSel.tyStringRecipeNm.sValue			:= p_tyMagRcpCurrRcp.sRcpNm;
	tyP0410MagSel.tyMagSel.tyNumMaxSlt.diValue				:= p_tyMagRcpCurrRcp.diTtlSlt;
	tyP0410MagSel.tyMagSel.tyNumSltToSltDist.diValue		:= p_tyMagRcpCurrRcp.diSltToSltInUM;
	tyP0410MagSel.tyMagSel.tyNumLifterMag1Slt1Pos.diValue	:= p_tyMagRcpCurrRcp.diMag1Slt1PosInUM;
	tyP0410MagSel.tyMagSel.tyNumLifterMag2Slt1Pos.diValue	:= p_tyMagRcpCurrRcp.diMag2Slt1PosInUM;
	tyP0410MagSel.tyMagSel.tyNumLifterMag3Slt1Pos.diValue	:= p_tyMagRcpCurrRcp.diMag3Slt1PosInUM;
	tyP0410MagSel.tyMagSel.tyNumTravPosMag1.diValue			:= p_tyMagRcpCurrRcp.diMag1TravPosInUM;
	tyP0410MagSel.tyMagSel.tyNumTravPosMag2.diValue			:= p_tyMagRcpCurrRcp.diMag2TravPosInUM;
	tyP0410MagSel.tyMagSel.tyNumTravPosMag3.diValue			:= p_tyMagRcpCurrRcp.diMag3TravPosInUM;
	tyP0410MagSel.tyMagSel.tyTxtMagModel.usiValueIdx		:= p_tyMagRcpCurrRcp.usiMagModel;
	tyP0410MagSel.tyMagSel.tyNumMagMaxBrdWidth.diValue		:= p_tyMagRcpCurrRcp.diMagMaxBrdWidth;
	tyP0410MagSel.tyMagSel.tyBtnMagHeightChkEn.bValue		:= p_tyMagRcpCurrRcp.bMagHeightChkEn;
	tyP0410MagSel.tyMagSel.tyBtnSafetyBar.bValue			:= p_tyMagRcpCurrRcp.bSafetyBarDisabled;

	tyP0410MagSel.tyMagSel.tyBtnSafetyBar.uiRtStat.0		:= NOT(p_tyNtParamCurr.bProjMagSafetyBarPrep);
	tyP0410MagSel.tyMagDet.tyBtnSafetyBar.uiRtStat.0		:= NOT(p_tyNtParamCurr.bProjMagSafetyBarPrep);

	tyP0410MagSel.tyMagSel.tyBtnMagHeightChkEn.uiRtStat.0	:= NOT(p_tyNtParamCurr.bProjMagHeightChkPrep);
	tyP0410MagSel.tyMagDet.tyBtnMagHeightChkEn.uiRtStat.0	:= NOT(p_tyNtParamCurr.bProjMagHeightChkPrep);

	tyP0410MagSel.tyMagSel.tyBitmapBrder.uiRtStat.0			:= NOT(p_tyNtParamCurr.bProjMagSafetyBarPrep OR
																	p_tyNtParamCurr.bProjMagHeightChkPrep);
END_ACTION
```

#### Act_Main_P0800.st
```iecst
ACTION Act_Main_P0800:

	//Display
	tyP0800MagInfo.tyMagInfo2.tyLyr.uiRtStat.0	:= NOT(p_tyNtParamCurr.eProjMag = ULMagTriple);

	tyP0800MagInfo.tyMagInfo1.tyBtnMag1SetFull.uiRtStat.0 := p_tyNtParamCurr.bProjLifterMagPlatform;
	tyP0800MagInfo.tyMagInfo1.tyBtnMag2SetFull.uiRtStat.0 := p_tyNtParamCurr.bProjLifterMagPlatform;
	tyP0800MagInfo.tyMagInfo2.tyBtnMag3SetFull.uiRtStat.0 := p_tyNtParamCurr.bProjLifterMagPlatform;

	tyP0800MagInfo.tyMagInfo1.tyBtnMag1SetFull.uiMaskRtStat.0 := p_tyNtParamCurr.bProjLifterMagPlatform;
	tyP0800MagInfo.tyMagInfo1.tyBtnMag2SetFull.uiMaskRtStat.0 := p_tyNtParamCurr.bProjLifterMagPlatform;
	tyP0800MagInfo.tyMagInfo2.tyBtnMag3SetFull.uiMaskRtStat.0 := p_tyNtParamCurr.bProjLifterMagPlatform;

END_ACTION
```

#### Act_Main_P0850.st
```iecst
ACTION Act_Main_P0850:

	//Display
	tyP0850OvenInfo.tyCom.tyBtnOvenB.uiRtStat.0	:= NOT p_tyNtParamCurr.bProjLaneBPrep;

	IF p_tyNtParamCurr.bMagAutoVerifyPrep=FALSE THEN
		tyP0850OvenInfo.tyCom.tyBitmapMc.uiValueIdx := 0;
	ELSE
		tyP0850OvenInfo.tyCom.tyBitmapMc.uiValueIdx := 20;
	END_IF

END_ACTION
```

#### Act_Main_P0900.st
```iecst
ACTION Act_Main_P0900:

	//Display
	tyP0900GenIn.tyGenIn2.tyLyr.uiRtStat.0	:= NOT p_tyNtParamCurr.bProjMagOrientChkSenPrep;

	tyP0900GenIn.tyGenIn1.tyBtnLifterTimingBeltSen.uiRtStat.0	:= p_tyNtParamCurr.tyDISettings.diLifterTimingBeltSen = 0;
	tyP0900GenIn.tyGenIn1.tyBtnLifterSafetyLmtSW1.uiRtStat.0	:= p_tyNtParamCurr.tyDISettings.diLifterSafetyLmtSW1 = 0;
	tyP0900GenIn.tyGenIn1.tyBtnLifterSafetyLmtSW2.uiRtStat.0	:= p_tyNtParamCurr.tyDISettings.diLifterSafetyLmtSW2 = 0;
	tyP0900GenIn.tyGenIn1.tyBtnMag3PresentSen.uiRtStat.0		:= NOT(p_tyNtParamCurr.eProjMag = ULMagTriple);
	tyP0900GenIn.tyGenIn1.tyBtnOvenInfeedSigA.uiRtStat.0		:= NOT(p_tyNtParamCurr.bOvenInfoPrep AND p_tyNtParamCurr.bOvenInfoExtdPrep);
	tyP0900GenIn.tyGenIn1.tyBtnOvenInfeedSigB.uiRtStat.0		:= NOT(p_tyNtParamCurr.bOvenInfoPrep AND p_tyNtParamCurr.bOvenInfoExtdPrep AND p_tyNtParamCurr.bProjLaneBPrep);
	tyP0900GenIn.tyGenIn1.tyBtnMagWidthChk.uiRtStat.0 			:= p_tyNtParamCurr.tyDISettings.diMagWidthChkSen = 0;

	tyP0900GenIn.tyGenIn2.tyBtnMag1OrientationChkSen1.uiRtStat.0	:= p_tyNtParamCurr.tyDISettings.diMag1OrientChkSen1 = 0;
	tyP0900GenIn.tyGenIn2.tyBtnMag2OrientationChkSen1.uiRtStat.0	:= p_tyNtParamCurr.tyDISettings.diMag2OrientChkSen1 = 0;
	tyP0900GenIn.tyGenIn2.tyBtnMag3OrientationChkSen1.uiRtStat.0	:= p_tyNtParamCurr.tyDISettings.diMag3OrientChkSen1 = 0;
	tyP0900GenIn.tyGenIn2.tyBtnMag1OrientationChkSen2.uiRtStat.0	:= p_tyNtParamCurr.tyDISettings.diMag1OrientChkSen2 = 0;
	tyP0900GenIn.tyGenIn2.tyBtnMag2OrientationChkSen2.uiRtStat.0	:= p_tyNtParamCurr.tyDISettings.diMag2OrientChkSen2 = 0;
	tyP0900GenIn.tyGenIn2.tyBtnMag3OrientationChkSen2.uiRtStat.0	:= p_tyNtParamCurr.tyDISettings.diMag3OrientChkSen2 = 0;
	tyP0900GenIn.tyGenIn2.tyBtnMag1HeightSen.uiRtStat.0				:= p_tyNtParamCurr.tyDISettings.diHighMagDetSen1 = 0;
	tyP0900GenIn.tyGenIn2.tyBtnMag2HeightSen.uiRtStat.0				:= p_tyNtParamCurr.tyDISettings.diHighMagDetSen2 = 0;
	tyP0900GenIn.tyGenIn2.tyBtnMag3HeightSen.uiRtStat.0				:= p_tyNtParamCurr.tyDISettings.diHighMagDetSen3 = 0;

	tyP0900GenIn.tyGenIn3.tyLyr.uiRtStat.0						:= NOT p_tyNtParamCurr.bCurtainSenPrep;

END_ACTION
```

#### Act_Main_P0910.st
```iecst
ACTION Act_Main_P0910:

	//Display
	tyP0910GenOut.tyGenOut.tyBtnBuzzer.uiRtStat.0	:= p_tyNtParamCurr.tyDOSettings.diBuzzer = 0;

	tyP0910GenOut.tyOven.tyLyr.uiRtStat.0	:= NOT p_tyNtParamCurr.bOvenInfoPrep;

	tyP0910GenOut.tyGenOutCurtainSen.tyLyr.uiRtStat.0	:= NOT p_tyNtParamCurr.bCurtainSenPrep;

	tyP0910GenOut.tyOven.tyBtnOvenInfoB.uiRtStat.0	:= NOT p_tyNtParamCurr.bProjLaneBPrep;

	tyP0910GenOut.tyMagAW.tyLyr12.uiRtStat.0	:= NOT p_tyNtParamCurr.bProjMagAWPrep;

	tyP0910GenOut.tyMagAW.tyLyr3.uiRtStat.0	:= NOT (p_tyNtParamCurr.bProjMagAWPrep AND p_tyNtParamCurr.eProjMag = ULMagTriple);

	tyP0910GenOut.tyMagAW.tyLyr4.uiRtStat.0	:= NOT (p_tyNtParamCurr.bProjMagAWPrep AND p_tyNtParamCurr.eProjMag = ULMagQuadruple);

	tyP0910GenOut.tyGenOut.tyBtnTLGreen.uiRtStat.0 :=  p_tyNtParamCurr.tyDOSettings.diTLGreen = 0;

	tyP0910GenOut.tyGenOut.tyBtnTLRed.uiRtStat.0 :=  p_tyNtParamCurr.tyDOSettings.diTLRed = 0;

	tyP0910GenOut.tyGenOut.tyBtnTLAmber.uiRtStat.0 :=  p_tyNtParamCurr.tyDOSettings.diTLAmber = 0;

	IF p_tyNtParamCurr.eCustomerReq = Siemens THEN
		tyP0910GenOut.tyGenOut.tyBtnTLAmber.usiTxtIdx := tyP0910GenOut.tyGenOut.tyBtnTLAmber.usiTxtIdx + 2 ;//White
	END_IF

END_ACTION
```

#### Act_Main_P0920.st
```iecst
ACTION Act_Main_P0920:

	//Machine Bitmap
	IF p_tyNtParamCurr.eProjMag = ULMagTriple AND p_tyNtParamCurr.bProjLifterMagPlatform AND p_tyNtParamCurr.bUIConvDirRL THEN
		tyP0920MtrNPneuCtrl.tyMtrNPneuCtrl.tyBtnAW.uiBitmapIdx				:= 500;
		tyP0920MtrNPneuCtrl.tyMtrNPneuCtrl.tyBtnLifter.uiBitmapIdx			:= 800;
		tyP0920MtrNPneuCtrl.tyMtrNPneuCtrl.tyBtnTrav.uiBitmapIdx			:= 800;
		tyP0920MtrNPneuCtrl.tyMtrNPneuCtrl.tyBtnPusherConv.uiBitmapIdx		:= 500;
		tyP0920MtrNPneuCtrl.tyMtrNPneuCtrlPneu.tyBtnShutter.uiBitmapIdx		:= 800;
		tyP0920MtrNPneuCtrl.tyMtrNPneuCtrl.tyBtnAWPushPul.uiBitmapIdx		:= 0;

	ELSIF p_tyNtParamCurr.eProjMag = ULMagDual AND p_tyNtParamCurr.bProjLifterMagPlatform AND p_tyNtParamCurr.bUIConvDirRL THEN
		tyP0920MtrNPneuCtrl.tyMtrNPneuCtrl.tyBtnAW.uiBitmapIdx				:= 500;
		tyP0920MtrNPneuCtrl.tyMtrNPneuCtrl.tyBtnLifter.uiBitmapIdx			:= 700;
		tyP0920MtrNPneuCtrl.tyMtrNPneuCtrl.tyBtnTrav.uiBitmapIdx			:= 700;
		tyP0920MtrNPneuCtrl.tyMtrNPneuCtrl.tyBtnPusherConv.uiBitmapIdx		:= 500;
		tyP0920MtrNPneuCtrl.tyMtrNPneuCtrlPneu.tyBtnShutter.uiBitmapIdx		:= 700;
		tyP0920MtrNPneuCtrl.tyMtrNPneuCtrl.tyBtnAWPushPul.uiBitmapIdx		:= 0;

	ELSIF p_tyNtParamCurr.eProjMag = ULMagTriple AND p_tyNtParamCurr.bProjLifterMagPlatform AND p_tyNtParamCurr.bUIConvDirRL = FALSE THEN
		tyP0920MtrNPneuCtrl.tyMtrNPneuCtrl.tyBtnAW.uiBitmapIdx				:= 500;
		tyP0920MtrNPneuCtrl.tyMtrNPneuCtrl.tyBtnLifter.uiBitmapIdx			:= 500;
		tyP0920MtrNPneuCtrl.tyMtrNPneuCtrl.tyBtnTrav.uiBitmapIdx			:= 500;
		tyP0920MtrNPneuCtrl.tyMtrNPneuCtrl.tyBtnPusherConv.uiBitmapIdx		:= 500;
		tyP0920MtrNPneuCtrl.tyMtrNPneuCtrlPneu.tyBtnShutter.uiBitmapIdx		:= 500;
		tyP0920MtrNPneuCtrl.tyMtrNPneuCtrl.tyBtnAWPushPul.uiBitmapIdx		:= 0;

	ELSIF p_tyNtParamCurr.eProjMag = ULMagDual AND p_tyNtParamCurr.bProjLifterMagPlatform AND p_tyNtParamCurr.bUIConvDirRL = FALSE
		AND p_tyNtParamCurr.bProjMagConvLane1Prep THEN
		tyP0920MtrNPneuCtrl.tyMtrNPneuCtrl.tyBtnAW.uiBitmapIdx				:= 500;//50
		tyP0920MtrNPneuCtrl.tyMtrNPneuCtrl.tyBtnLifter.uiBitmapIdx			:= 900;//51
		tyP0920MtrNPneuCtrl.tyMtrNPneuCtrl.tyBtnLifter2.uiBitmapIdx			:= 901;
		tyP0920MtrNPneuCtrl.tyMtrNPneuCtrl.tyBtnMag1Conv.uiBitmapIdx		:= 902;
		tyP0920MtrNPneuCtrl.tyMtrNPneuCtrl.tyBtnTrav.uiBitmapIdx			:= 600;//52
		tyP0920MtrNPneuCtrl.tyMtrNPneuCtrl.tyBtnPusherConv.uiBitmapIdx		:= 500;//53
		tyP0920MtrNPneuCtrl.tyMtrNPneuCtrl.tyBtnLifterConv.uiBitmapIdx		:= 900;
		tyP0920MtrNPneuCtrl.tyMtrNPneuCtrl.tyBtnLifterConv2.uiBitmapIdx		:= 901;
		tyP0920MtrNPneuCtrl.tyMtrNPneuCtrlPneu.tyBtnShutter.uiBitmapIdx		:= 900; //54
		tyP0920MtrNPneuCtrl.tyMtrNPneuCtrl.tyBtnAWPushPul.uiBitmapIdx		:= 0;

	ELSIF p_tyNtParamCurr.eProjMag = ULMagDual AND p_tyNtParamCurr.bProjLifterMagPlatform AND p_tyNtParamCurr.bUIConvDirRL = FALSE THEN
		tyP0920MtrNPneuCtrl.tyMtrNPneuCtrl.tyBtnAW.uiBitmapIdx				:= 500;
		tyP0920MtrNPneuCtrl.tyMtrNPneuCtrl.tyBtnLifter.uiBitmapIdx			:= 600;
		tyP0920MtrNPneuCtrl.tyMtrNPneuCtrl.tyBtnTrav.uiBitmapIdx			:= 600;
		tyP0920MtrNPneuCtrl.tyMtrNPneuCtrl.tyBtnPusherConv.uiBitmapIdx		:= 500;
		tyP0920MtrNPneuCtrl.tyMtrNPneuCtrlPneu.tyBtnShutter.uiBitmapIdx		:= 600;
		tyP0920MtrNPneuCtrl.tyMtrNPneuCtrl.tyBtnAWPushPul.uiBitmapIdx		:= 0;

	ELSIF p_tyNtParamCurr.eProjMag = ULMagTriple AND p_tyNtParamCurr.bMagAutoVerifyPrep = FALSE THEN
		tyP0920MtrNPneuCtrl.tyMtrNPneuCtrl.tyBtnAW.uiBitmapIdx				:= 100;
		tyP0920MtrNPneuCtrl.tyMtrNPneuCtrl.tyBtnLifter.uiBitmapIdx			:= 100;
		tyP0920MtrNPneuCtrl.tyMtrNPneuCtrl.tyBtnTrav.uiBitmapIdx			:= 100;
		tyP0920MtrNPneuCtrl.tyMtrNPneuCtrl.tyBtnPusherConv.uiBitmapIdx		:= 100;
		tyP0920MtrNPneuCtrl.tyMtrNPneuCtrl.tyBtnMag1Conv.uiBitmapIdx		:= 106;
		tyP0920MtrNPneuCtrl.tyMtrNPneuCtrl.tyBtnMag2Conv.uiBitmapIdx		:= 100;
		tyP0920MtrNPneuCtrl.tyMtrNPneuCtrl.tyBtnMag3Conv.uiBitmapIdx		:= 100;
		tyP0920MtrNPneuCtrl.tyMtrNPneuCtrlPneu.tyBtnShutter.uiBitmapIdx	:= 100;
		tyP0920MtrNPneuCtrl.tyMtrNPneuCtrlPneu.tyBtnSafetyBar.usiBitmapIdx	:= 100;
		tyP0920MtrNPneuCtrl.tyMtrNPneuCtrl.tyBtnAWPushPul.uiBitmapIdx		:= 0;
	ELSIF p_tyNtParamCurr.eProjMag = ULMagDual AND p_tyNtParamCurr.bMagAutoVerifyPrep = TRUE AND p_tyNtParamCurr.bProjMagAWPrep = FALSE THEN
		tyP0920MtrNPneuCtrl.tyMtrNPneuCtrl.tyBtnAW.uiBitmapIdx				:= 200;
		tyP0920MtrNPneuCtrl.tyMtrNPneuCtrl.tyBtnLifter.uiBitmapIdx			:= 200;
		tyP0920MtrNPneuCtrl.tyMtrNPneuCtrl.tyBtnTrav.uiBitmapIdx			:= 200;
		tyP0920MtrNPneuCtrl.tyMtrNPneuCtrl.tyBtnMag1Conv.uiBitmapIdx		:= 154;
		tyP0920MtrNPneuCtrl.tyMtrNPneuCtrl.tyBtnMag2Conv.uiBitmapIdx		:= 200;
		tyP0920MtrNPneuCtrl.tyMtrNPneuCtrl.tyBtnMag3Conv.uiBitmapIdx		:= 200;
		tyP0920MtrNPneuCtrl.tyMtrNPneuCtrlPneu.tyBtnStopper.uiBitmapIdx	:= 100;
		tyP0920MtrNPneuCtrl.tyMtrNPneuCtrlPneu.tyBtnShutter.uiBitmapIdx	:= 200;
		tyP0920MtrNPneuCtrl.tyMtrNPneuCtrlPneu.tyBtnSafetyBar.usiBitmapIdx	:= 100;
		tyP0920MtrNPneuCtrl.tyMtrNPneuCtrl.tyBtnAWPushPul.uiBitmapIdx		:= 0;
	ELSIF p_tyNtParamCurr.eProjMag = ULMagTriple AND p_tyNtParamCurr.bMagAutoVerifyPrep = TRUE AND p_tyNtParamCurr.bProjMagAWPrep THEN
		tyP0920MtrNPneuCtrl.tyMtrNPneuCtrl.tyBtnAW.uiBitmapIdx				:= 200;
		tyP0920MtrNPneuCtrl.tyMtrNPneuCtrl.tyBtnLifter.uiBitmapIdx			:= 200;
		tyP0920MtrNPneuCtrl.tyMtrNPneuCtrl.tyBtnTrav.uiBitmapIdx			:= 200;
		tyP0920MtrNPneuCtrl.tyMtrNPneuCtrl.tyBtnMag1Conv.uiBitmapIdx		:= 106;
		tyP0920MtrNPneuCtrl.tyMtrNPneuCtrl.tyBtnMag2Conv.uiBitmapIdx		:= 200;
		tyP0920MtrNPneuCtrl.tyMtrNPneuCtrl.tyBtnMag3Conv.uiBitmapIdx		:= 200;
		tyP0920MtrNPneuCtrl.tyMtrNPneuCtrlPneu.tyBtnStopper.uiBitmapIdx	:= 100;
		tyP0920MtrNPneuCtrl.tyMtrNPneuCtrlPneu.tyBtnShutter.uiBitmapIdx	:= 200;
		tyP0920MtrNPneuCtrl.tyMtrNPneuCtrl.tyBtnMagAW.uiBitmapIdx			:= 0;
		tyP0920MtrNPneuCtrl.tyMtrNPneuCtrlPneu.tyBtnSafetyBar.usiBitmapIdx	:= 100;
		tyP0920MtrNPneuCtrl.tyMtrNPneuCtrl.tyBtnAWPushPul.uiBitmapIdx		:= 0;
	ELSIF p_tyNtParamCurr.eProjMag = ULMagDual AND p_tyNtParamCurr.bMagAutoVerifyPrep = TRUE AND p_tyNtParamCurr.bProjMagAWPrep THEN
		tyP0920MtrNPneuCtrl.tyMtrNPneuCtrl.tyBtnAW.uiBitmapIdx				:= 300;
		tyP0920MtrNPneuCtrl.tyMtrNPneuCtrl.tyBtnLifter.uiBitmapIdx			:= 300;
		tyP0920MtrNPneuCtrl.tyMtrNPneuCtrl.tyBtnTrav.uiBitmapIdx			:= 300;
		tyP0920MtrNPneuCtrl.tyMtrNPneuCtrl.tyBtnMag1Conv.uiBitmapIdx		:= 298;
		tyP0920MtrNPneuCtrl.tyMtrNPneuCtrl.tyBtnMag2Conv.uiBitmapIdx		:= 300;
		tyP0920MtrNPneuCtrl.tyMtrNPneuCtrl.tyBtnMag3Conv.uiBitmapIdx		:= 300;
		tyP0920MtrNPneuCtrl.tyMtrNPneuCtrlPneu.tyBtnStopper.uiBitmapIdx	:= 100;
		tyP0920MtrNPneuCtrl.tyMtrNPneuCtrlPneu.tyBtnShutter.uiBitmapIdx	:= 300;
		tyP0920MtrNPneuCtrl.tyMtrNPneuCtrl.tyBtnMagAW.uiBitmapIdx			:= 100;
		tyP0920MtrNPneuCtrl.tyMtrNPneuCtrlPneu.tyBtnSafetyBar.uiBitmapIdx	:= 100;
		tyP0920MtrNPneuCtrl.tyMtrNPneuCtrl.tyBtnAWPushPul.usiBitmapIdx		:= 0;
	ELSIF p_tyNtParamCurr.eProjMag = ULMagDual AND p_tyNtParamCurr.bMagAutoVerifyPrep = FALSE AND p_tyNtParamCurr.bProjMagAWPrep = FALSE THEN
		tyP0920MtrNPneuCtrl.tyMtrNPneuCtrl.tyBtnAW.uiBitmapIdx				:= 300;
		tyP0920MtrNPneuCtrl.tyMtrNPneuCtrl.tyBtnLifter.uiBitmapIdx			:= 300;
		tyP0920MtrNPneuCtrl.tyMtrNPneuCtrl.tyBtnTrav.uiBitmapIdx			:= 300;
		tyP0920MtrNPneuCtrl.tyMtrNPneuCtrl.tyBtnMag1Conv.uiBitmapIdx		:= 298;
		tyP0920MtrNPneuCtrl.tyMtrNPneuCtrl.tyBtnMag2Conv.uiBitmapIdx		:= 300;
		tyP0920MtrNPneuCtrl.tyMtrNPneuCtrl.tyBtnMag3Conv.uiBitmapIdx		:= 300;
		tyP0920MtrNPneuCtrl.tyMtrNPneuCtrlPneu.tyBtnStopper.uiBitmapIdx	:= 100;
		tyP0920MtrNPneuCtrl.tyMtrNPneuCtrlPneu.tyBtnShutter.uiBitmapIdx	:= 300;
		tyP0920MtrNPneuCtrl.tyMtrNPneuCtrl.tyBtnMagAW.uiBitmapIdx			:= 100;
		tyP0920MtrNPneuCtrl.tyMtrNPneuCtrlPneu.tyBtnSafetyBar.usiBitmapIdx	:= 100;
		tyP0920MtrNPneuCtrl.tyMtrNPneuCtrl.tyBtnAWPushPul.uiBitmapIdx		:= 0;
	ELSE
		tyP0920MtrNPneuCtrl.tyMtrNPneuCtrl.tyBtnAW.uiBitmapIdx				:= 0;
		tyP0920MtrNPneuCtrl.tyMtrNPneuCtrl.tyBtnLifter.uiBitmapIdx			:= 0;
		tyP0920MtrNPneuCtrl.tyMtrNPneuCtrl.tyBtnTrav.uiBitmapIdx			:= 0;
		tyP0920MtrNPneuCtrl.tyMtrNPneuCtrl.tyBtnPusherConv.uiBitmapIdx		:= 0;
		tyP0920MtrNPneuCtrl.tyMtrNPneuCtrl.tyBtnMag1Conv.uiBitmapIdx		:= 0;
		tyP0920MtrNPneuCtrl.tyMtrNPneuCtrl.tyBtnMag2Conv.uiBitmapIdx		:= 0;
		tyP0920MtrNPneuCtrl.tyMtrNPneuCtrl.tyBtnMag3Conv.uiBitmapIdx		:= 0;
		tyP0920MtrNPneuCtrl.tyMtrNPneuCtrlPneu.tyBtnShutter.uiBitmapIdx	:= 0;
		tyP0920MtrNPneuCtrl.tyMtrNPneuCtrlPneu.tyBtnStopper.uiBitmapIdx	:= 0;
		tyP0920MtrNPneuCtrl.tyMtrNPneuCtrlPneu.tyBtnSafetyBar.usiBitmapIdx	:= 100;
		tyP0920MtrNPneuCtrl.tyMtrNPneuCtrl.tyBtnAWPushPul.uiBitmapIdx		:= 0;
	END_IF

	//Auto Width
	tyP0920MtrNPneuCtrl.tyMtrNPneuCtrl.tyBtnAW.uiRtStat.0	:= NOT p_tyNtParamCurr.bAWPrep;

	//Magazine Auto Width
	tyP0920MtrNPneuCtrl.tyMtrNPneuCtrl.tyBtnMagAW.uiRtStat.0	:= NOT p_tyNtParamCurr.bProjMagAWPrep;

	//Pneumatic
	tyP0920MtrNPneuCtrl.tyMtrNPneuCtrlPneu.tyLyr.uiRtStat.0	:= NOT(p_tyNtParamCurr.bProjInletShutPrep OR p_tyNtParamCurr.bProjOutletShutPrep
																OR p_tyNtParamCurr.bProjStopperAPrep OR p_tyNtParamCurr.bProjStopperBPrep);

	//Shutter
	tyP0920MtrNPneuCtrl.tyMtrNPneuCtrlPneu.tyBtnShutter.uiRtStat.0  := NOT(p_tyNtParamCurr.bProjInletShutPrep OR p_tyNtParamCurr.bProjOutletShutPrep);

	//Stopper
	tyP0920MtrNPneuCtrl.tyMtrNPneuCtrlPneu.tyBtnStopper.uiRtStat.0	:= NOT(p_tyNtParamCurr.bProjStopperAPrep OR p_tyNtParamCurr.bProjStopperBPrep OR p_tyNtParamCurr.bProjInletStopperPrep);

	//Magazine Conveyor
	tyP0920MtrNPneuCtrl.tyMtrNPneuCtrl.tyBtnMag1Conv.uiRtStat.0	:= NOT((p_tyNtParamCurr.bProjMag1ConvPrep OR p_tyNtParamCurr.bProjMag2ConvPrep OR p_tyNtParamCurr.bProjMag3ConvPrep OR
																	p_tyNtParamCurr.bProjMagConvLane1Prep OR p_tyNtParamCurr.bProjMagConvLane2Prep) AND p_tyNtParamCurr.bProjLifTravMnlLoad= FALSE);
//	tyP0920MtrNPneuCtrl.tyMtrNPneuCtrl.tyBtnMag1Conv.uiRtStat.0	:= NOT(NOT (p_tyNtParamCurr.bProjMag1ConvPrep AND p_tyNtParamCurr.bProjMag2ConvPrep AND p_tyNtParamCurr.bProjMag3ConvPrep)XOR
//																	NOT (p_tyNtParamCurr.bProjMagConvLane1Prep AND p_tyNtParamCurr.bProjMagConvLane2Prep)));
//	tyP0920MtrNPneuCtrl.tyMtrNPneuCtrl.tyBtnMag2Conv.uiRtStat.0	:= NOT p_tyNtParamCurr.bProjMag2ConvPrep;
//	tyP0920MtrNPneuCtrl.tyMtrNPneuCtrl.tyBtnMag3Conv.uiRtStat.0	:= NOT(p_tyNtParamCurr.bProjMag3ConvPrep AND (p_tyNtParamCurr.eProjMag = ULMagTriple));

	//Safety Bar
	tyP0920MtrNPneuCtrl.tyMtrNPneuCtrlPneu.tyBtnSafetyBar.uiRtStat.0	:= NOT p_tyNtParamCurr.bProjMagSafetyBarPrep;
	//Pusher Auto Width
	tyP0920MtrNPneuCtrl.tyMtrNPneuCtrl.tyBtnAWPushPul.uiRtStat.0	:= NOT p_tyNtParamCurr.bAWPusherPrep;
	//Lifter2
	tyP0920MtrNPneuCtrl.tyMtrNPneuCtrl.tyBtnLifter2.uiRtStat.0	:= NOT p_tyNtParamCurr.bProjLifter2Prep;
	tyP0920MtrNPneuCtrl.tyMtrNPneuCtrl.tyBtnLifter.uiRtStat.0	:= NOT p_tyNtParamCurr.bProjLifter2Prep;
	tyP0920MtrNPneuCtrl.tyMtrNPneuCtrl.tyBtnLifterBigBtn.uiRtStat.0	:= p_tyNtParamCurr.bProjLifter2Prep;
	//Lifter Conveyor
	tyP0920MtrNPneuCtrl.tyMtrNPneuCtrl.tyBtnLifterConv.uiRtStat.0	:= NOT p_tyNtParamCurr.bProjMagConvLane1Prep;
	tyP0920MtrNPneuCtrl.tyMtrNPneuCtrl.tyBtnLifterConv2.uiRtStat.0	:= NOT p_tyNtParamCurr.bProjMagConvLane2Prep;

END_ACTION
```

#### Act_Main_P0921.st
```iecst
ACTION Act_Main_P0921:

	//Display
	tyP0921InletNOutletShutter.tyInletShutterCom.tyLyr.uiRtStat.0	:= NOT(p_tyNtParamCurr.bProjInletShutPrep);
	tyP0921InletNOutletShutter.tyInletShutterDC.tyLyr.uiRtStat.0	:= TRUE;
	tyP0921InletNOutletShutter.tyInletShutterFB.tyLyr.uiRtStat.0	:= NOT(p_tyNtParamCurr.bProjInletShutPrep);

	tyP0921InletNOutletShutter.tyOutletShutterCom.tyLyr.uiRtStat.0	:= NOT(p_tyNtParamCurr.bProjOutletShutPrep);
	tyP0921InletNOutletShutter.tyOutletShutterDC.tyLyr.uiRtStat.0	:= TRUE;
	tyP0921InletNOutletShutter.tyOutletShutterFB.tyLyr.uiRtStat.0	:= NOT(p_tyNtParamCurr.bProjOutletShutPrep);

END_ACTION
```

#### Act_Main_P0922.st
```iecst
ACTION Act_Main_P0922:

	//Display
	tyP0922Stopper.tyStopperACom.tyLyr.uiRtStat.0	:= NOT(p_tyNtParamCurr.bProjStopperAPrep);
	tyP0922Stopper.tyStopperADC.tyLyr.uiRtStat.0	:= TRUE;
	tyP0922Stopper.tyStopperAFB.tyLyr.uiRtStat.0	:= NOT(p_tyNtParamCurr.bProjStopperAPrep);

	tyP0922Stopper.tyStopperBCom.tyLyr.uiRtStat.0	:= NOT(p_tyNtParamCurr.bProjStopperBPrep);
	tyP0922Stopper.tyStopperBDC.tyLyr.uiRtStat.0	:= TRUE;
	tyP0922Stopper.tyStopperBFB.tyLyr.uiRtStat.0	:= NOT(p_tyNtParamCurr.bProjStopperBPrep);

	//Inlet Stopper
	tyP0922Stopper.tyInStopperCom.tyLyr.uiRtStat.0	:= NOT(p_tyNtParamCurr.bProjInletStopperPrep);
	tyP0922Stopper.tyInStopperDC.tyLyr.uiRtStat.0	:= TRUE;
	tyP0922Stopper.tyInStopperFB.tyLyr.uiRtStat.0	:= NOT(p_tyNtParamCurr.bProjInletStopperPrep);

END_ACTION
```

#### Act_Main_P0923.st
```iecst
ACTION Act_Main_P0923:

	//Display

END_ACTION
```

#### Act_Main_P0928.st
```iecst
ACTION Act_Main_P0928:

	//Display //Sensor
	tyP0928MagConv.tyCom.tyBtnTopEntSen.uiRtStat.0	:= p_tyNtParamCurr.tyDISettings.diInMagConvEntSen = 0;
	tyP0928MagConv.tyCom.tyBtnTopMidSen.uiRtStat.0	:= p_tyNtParamCurr.tyDISettings.diInMagConvMidSen = 0;
	tyP0928MagConv.tyCom.tyBtnTopExtSen.uiRtStat.0	:= p_tyNtParamCurr.tyDISettings.diInMagConvExtSen = 0;
	tyP0928MagConv.tyCom.tyBtnBtmEntSen.uiRtStat.0	:= p_tyNtParamCurr.tyDISettings.diOutMagConvEntSen = 0;
	tyP0928MagConv.tyCom.tyBtnBtmMidSen.uiRtStat.0	:= p_tyNtParamCurr.tyDISettings.diOutMagConvMidSen = 0;
	tyP0928MagConv.tyCom.tyBtnBtmExtSen.uiRtStat.0	:= p_tyNtParamCurr.tyDISettings.diOutMagConvExtSen = 0;
	//Display //Stopper
	tyP0928MagConv.tyCom.tyBtnTopEntStprExtRS.uiRtStat.0	:= TRUE;
	tyP0928MagConv.tyCom.tyBtnTopEntStprRetRS.uiRtStat.0	:= TRUE;
	tyP0928MagConv.tyCom.tyBtnTopMidStprExtRS.uiRtStat.0	:= TRUE;
	tyP0928MagConv.tyCom.tyBtnTopMidStprRetRS.uiRtStat.0	:= TRUE;
	tyP0928MagConv.tyCom.tyBtnTopExtStprExtRS.uiRtStat.0	:= TRUE;
	tyP0928MagConv.tyCom.tyBtnTopExtStprRetRS.uiRtStat.0	:= TRUE;

	tyP0928MagConv.tyCom.tyBtnBtmMidStprExtRS.uiRtStat.0	:= TRUE;
	tyP0928MagConv.tyCom.tyBtnBtmMidStprRetRS.uiRtStat.0	:= TRUE;
	tyP0928MagConv.tyCom.tyBtnBtmExtStprExtRS.uiRtStat.0	:= TRUE;
	tyP0928MagConv.tyCom.tyBtnBtmExtStprRetRS.uiRtStat.0	:= TRUE;

	//control btn
	tyP0928MagConv.tyTopFB.tyBtnEntStprExt.uiRtStat := p_tyNtParamCurr.tyDOSettings.diEntTopStprUnblkCtrl = 0;
	tyP0928MagConv.tyTopDC.tyBtnEntStprExt.uiRtStat := p_tyNtParamCurr.tyDOSettings.diEntTopStprUnblkCtrl = 0;
	tyP0928MagConv.tyTopFB.tyBtnEntStprRet.uiRtStat := p_tyNtParamCurr.tyDOSettings.diEntTopStprUnblkCtrl = 0;
	tyP0928MagConv.tyTopDC.tyBtnEntStprRet.uiRtStat := p_tyNtParamCurr.tyDOSettings.diEntTopStprUnblkCtrl = 0;

END_ACTION
```

#### Act_Main_P0929.st
```iecst
ACTION Act_Main_P0929:

	//Display //Sensor
	tyP0929MagConv2.tyCom.tyBtnTopEntSen.uiRtStat.0	:= p_tyNtParamCurr.tyDISettings.diInMagConv2EntSen = 0;
	tyP0929MagConv2.tyCom.tyBtnTopMidSen.uiRtStat.0	:= p_tyNtParamCurr.tyDISettings.diInMagConv2MidSen = 0;
	tyP0929MagConv2.tyCom.tyBtnTopExtSen.uiRtStat.0	:= p_tyNtParamCurr.tyDISettings.diInMagConv2ExtSen = 0;
	tyP0929MagConv2.tyCom.tyBtnBtmEntSen.uiRtStat.0	:= p_tyNtParamCurr.tyDISettings.diOutMagConv2EntSen = 0;
	tyP0929MagConv2.tyCom.tyBtnBtmMidSen.uiRtStat.0	:= p_tyNtParamCurr.tyDISettings.diOutMagConv2MidSen = 0;
	tyP0929MagConv2.tyCom.tyBtnBtmExtSen.uiRtStat.0	:= p_tyNtParamCurr.tyDISettings.diOutMagConv2ExtSen = 0;
	//Display //Stopper
	tyP0929MagConv2.tyCom.tyBtnTopEntStprExtRS.uiRtStat.0	:= TRUE;
	tyP0929MagConv2.tyCom.tyBtnTopEntStprRetRS.uiRtStat.0	:= TRUE;
	tyP0929MagConv2.tyCom.tyBtnTopMidStprExtRS.uiRtStat.0	:= TRUE;
	tyP0929MagConv2.tyCom.tyBtnTopMidStprRetRS.uiRtStat.0	:= TRUE;
	tyP0929MagConv2.tyCom.tyBtnTopExtStprExtRS.uiRtStat.0	:= TRUE;
	tyP0929MagConv2.tyCom.tyBtnTopExtStprRetRS.uiRtStat.0	:= TRUE;

	tyP0929MagConv2.tyCom.tyBtnBtmMidStprExtRS.uiRtStat.0	:= TRUE;
	tyP0929MagConv2.tyCom.tyBtnBtmMidStprRetRS.uiRtStat.0	:= TRUE;
	tyP0929MagConv2.tyCom.tyBtnBtmExtStprExtRS.uiRtStat.0	:= TRUE;
	tyP0929MagConv2.tyCom.tyBtnBtmExtStprRetRS.uiRtStat.0	:= TRUE;

	//Control btn
	tyP0929MagConv2.tyTopFB.tyBtnEntStprExt.uiRtStat := p_tyNtParamCurr.tyDOSettings.diEntTopStprUnblkCtrl2 = 0;
	tyP0929MagConv2.tyTopDC.tyBtnEntStprExt.uiRtStat := p_tyNtParamCurr.tyDOSettings.diEntTopStprUnblkCtrl2 = 0;
	tyP0929MagConv2.tyTopFB.tyBtnEntStprRet.uiRtStat := p_tyNtParamCurr.tyDOSettings.diEntTopStprUnblkCtrl2 = 0;
	tyP0929MagConv2.tyTopDC.tyBtnEntStprRet.uiRtStat := p_tyNtParamCurr.tyDOSettings.diEntTopStprUnblkCtrl2 = 0;

END_ACTION
```

#### Act_Main_P0930.st
```iecst
ACTION Act_Main_P0930:

	//Display
	tyP0930MagConv1.tyCom.tyBtnMagAIVPosSen1.uiRtStat.0			:= p_tyNtParamCurr.tyDISettings.diMag1AIVInPosSen1 = 0;
	tyP0930MagConv1.tyCom.tyBtnMagAIVPosSen2.uiRtStat.0			:= p_tyNtParamCurr.tyDISettings.diMag1AIVInPosSen2 = 0;
	tyP0930MagConv1.tyCom.tyBtnMagOrientationChkSen1.uiRtStat.0	:= p_tyNtParamCurr.tyDISettings.diMag1OrientChkSen1 = 0;
	tyP0930MagConv1.tyCom.tyBtnMagOrientationChkSen2.uiRtStat.0	:= p_tyNtParamCurr.tyDISettings.diMag1OrientChkSen2 = 0;

	//Hide the following when in MagAutoVerify
	tyP0930MagConv1.tyCom.tyBtnRemoteClampRS.uiRtStat.0			:= p_tyNtParamCurr.tyDISettings.diMag1RemoteClampRS = 0;
	tyP0930MagConv1.tyCom.tyBtnRemoteUnclampRS.uiRtStat.0		:= p_tyNtParamCurr.tyDISettings.diMag1RemoteUnclampRS = 0 ;
	tyP0930MagConv1.tyCom.tyBtnFixedClampRS.uiRtStat.0			:= p_tyNtParamCurr.bMagAutoVerifyPrep;

	//Show the following in MagAutoVerify
//	tyP0930MagConv1.tyCom.tyBtnHeightSen.uiRtStat.0				:= NOT p_tyNtParamCurr.bMagAutoVerifyPrep;
	tyP0930MagConv1.tyCom.tyBtnCAB717Sen.uiRtStat.0				:= NOT p_tyNtParamCurr.bMagAutoVerifyPrep;
	tyP0930MagConv1.tyCom.tyBtnMagLargeSen.uiRtStat.0			:= NOT p_tyNtParamCurr.bMagAutoVerifyPrep;
	tyP0930MagConv1.tyCom.tyBtnMagSmallSen.uiRtStat.0			:= NOT p_tyNtParamCurr.bMagAutoVerifyPrep;
	tyP0930MagConv1.tyCom.tyBtnSelClampRS.uiRtStat.0			:= NOT p_tyNtParamCurr.bMagAutoVerifyPrep;
	tyP0930MagConv1.tyCom.tyBtnSelUnclampRS.uiRtStat.0			:= NOT p_tyNtParamCurr.bMagAutoVerifyPrep;
	tyP0930MagConv1.tyCom.tyBtnFixedUnclampRS.uiRtStat.0		:= NOT p_tyNtParamCurr.bMagAutoVerifyPrep;
	tyP0930MagConv1.tyCom.tyBtnMagDetectSen.uiRtStat.0			:= NOT p_tyNtParamCurr.bProjFixClprMagDetectSenPrep;
	//Show the MagHigh Sensor
	tyP0930MagConv1.tyCom.tyBtnHeightSen.uiRtStat.0				:= NOT p_tyNtParamCurr.bProjMagHeightChkPrep;

	IF p_tyNtParamCurr.bMagAutoVerifyPrep = FALSE THEN
		tyP0930MagConv1.tyDC.tyBtnFixedClamp.usiTxtIdx:= 6;
		tyP0930MagConv1.tyDC.tyBtnFixedUnclamp.usiTxtIdx:= 6;
		tyP0930MagConv1.tyDC.tyBtnRemoteClamp.usiTxtIdx:= 6;
		tyP0930MagConv1.tyDC.tyBtnRemoteUnclamp.usiTxtIdx:= 6;

		tyP0930MagConv1.tyFB.tyBtnFixedClamp.usiTxtIdx:= 6;
		tyP0930MagConv1.tyFB.tyBtnFixedUnclamp.usiTxtIdx:= 6;
		tyP0930MagConv1.tyFB.tyBtnRemoteClamp.usiTxtIdx:= 6;
		tyP0930MagConv1.tyFB.tyBtnRemoteUnclamp.usiTxtIdx:= 6;

		tyP0930MagConv1.tyCom.tyBtnFixedUnclampRS.usiTxtIdx:= 5;
		tyP0930MagConv1.tyCom.tyBtnFixedClampRS.usiTxtIdx:= 10;
		tyP0930MagConv1.tyCom.tyBtnRemoteUnclampRS.usiTxtIdx:= 4;

	ELSE IF p_tyNtParamCurr.bMagAutoVerifyPrep = TRUE THEN

		tyP0930MagConv1.tyDC.tyBtnFixedClamp.usiTxtIdx:= 6;
		tyP0930MagConv1.tyDC.tyBtnFixedUnclamp.usiTxtIdx:= 6;
		tyP0930MagConv1.tyDC.tyBtnRemoteClamp.usiTxtIdx:= 6;
		tyP0930MagConv1.tyDC.tyBtnRemoteUnclamp.usiTxtIdx:= 6;

		tyP0930MagConv1.tyFB.tyBtnFixedClamp.usiTxtIdx:= 6;
		tyP0930MagConv1.tyFB.tyBtnFixedUnclamp.usiTxtIdx:= 6;
		tyP0930MagConv1.tyFB.tyBtnRemoteClamp.usiTxtIdx:= 6;
		tyP0930MagConv1.tyFB.tyBtnRemoteUnclamp.usiTxtIdx:= 6;

		tyP0930MagConv1.tyCom.tyBtnFixedUnclampRS.usiTxtIdx:= 5;
		tyP0930MagConv1.tyCom.tyBtnRemoteUnclampRS.usiTxtIdx:= 4;
		END_IF
	END_IF

	IF p_tyNtParamCurr.bMagAutoVerifyPrep AND p_tyNtParamCurr.bProjMagAWPrep = FALSE THEN
		tyP0930MagConv1.tyCom.tyBitmapMc.uiValueIdx	:= 0;
	ELSIF p_tyNtParamCurr.bMagAutoVerifyPrep AND p_tyNtParamCurr.bProjMagAWPrep THEN
		tyP0930MagConv1.tyCom.tyBitmapMc.uiValueIdx	:= 3;
	ELSIF p_tyNtParamCurr.bMagAutoVerifyPrep = FALSE AND p_tyNtParamCurr.bProjMagAWPrep = FALSE AND p_tyNtParamCurr.bProjMagSafetyBarPrep = TRUE THEN
		tyP0930MagConv1.tyCom.tyBitmapMc.uiValueIdx	:= 201;
	ELSE
		tyP0930MagConv1.tyCom.tyBitmapMc.uiValueIdx	:= 233;
	END_IF

END_ACTION
```

#### Act_Main_P0931.st
```iecst
ACTION Act_Main_P0931:

	//Display
	tyP0931MagConv2.tyCom.tyBtnMagAIVPosSen1.uiRtStat.0			:= p_tyNtParamCurr.tyDISettings.diMag2AIVInPosSen1 = 0;
	tyP0931MagConv2.tyCom.tyBtnMagAIVPosSen2.uiRtStat.0			:= p_tyNtParamCurr.tyDISettings.diMag2AIVInPosSen2 = 0;
	tyP0931MagConv2.tyCom.tyBtnMagOrientationChkSen1.uiRtStat.0	:= p_tyNtParamCurr.tyDISettings.diMag2OrientChkSen1 = 0;
	tyP0931MagConv2.tyCom.tyBtnMagOrientationChkSen2.uiRtStat.0	:= p_tyNtParamCurr.tyDISettings.diMag2OrientChkSen2 = 0;

	//Hide the following when in MagAutoVerify
	tyP0931MagConv2.tyCom.tyBtnRemoteClampRS.uiRtStat.0			:= p_tyNtParamCurr.tyDISettings.diMag2RemoteClampRS = 0;
	tyP0931MagConv2.tyCom.tyBtnRemoteUnclampRS.uiRtStat.0		:=  p_tyNtParamCurr.tyDISettings.diMag1RemoteUnclampRS = 0 ;
	tyP0931MagConv2.tyCom.tyBtnFixedClampRS.uiRtStat.0			:= p_tyNtParamCurr.bMagAutoVerifyPrep;

//	tyP0931MagConv2.tyCom.tyBtnHeightSen.uiRtStat.0				:= NOT p_tyNtParamCurr.bMagAutoVerifyPrep;
	tyP0931MagConv2.tyCom.tyBtnCAB717Sen.uiRtStat.0				:= NOT p_tyNtParamCurr.bMagAutoVerifyPrep;
	tyP0931MagConv2.tyCom.tyBtnMagLargeSen.uiRtStat.0			:= NOT p_tyNtParamCurr.bMagAutoVerifyPrep;
	tyP0931MagConv2.tyCom.tyBtnMagSmallSen.uiRtStat.0			:= NOT p_tyNtParamCurr.bMagAutoVerifyPrep;
	tyP0931MagConv2.tyCom.tyBtnSelClampRS.uiRtStat.0			:= NOT p_tyNtParamCurr.bMagAutoVerifyPrep;
	tyP0931MagConv2.tyCom.tyBtnSelUnclampRS.uiRtStat.0			:= NOT p_tyNtParamCurr.bMagAutoVerifyPrep;
	tyP0931MagConv2.tyCom.tyBtnFixedUnclampRS.uiRtStat.0		:= NOT p_tyNtParamCurr.bMagAutoVerifyPrep;
	tyP0931MagConv2.tyCom.tyBtnMagDetectSen.uiRtStat.0			:= NOT p_tyNtParamCurr.bProjFixClprMagDetectSenPrep;

	tyP0931MagConv2.tyCom.tyBtnHeightSen.uiRtStat.0				:= NOT p_tyNtParamCurr.bProjMagHeightChkPrep;

	IF p_tyNtParamCurr.bMagAutoVerifyPrep = FALSE THEN
		tyP0931MagConv2.tyDC.tyBtnFixedClamp.usiTxtIdx:= 6;
		tyP0931MagConv2.tyDC.tyBtnFixedUnclamp.usiTxtIdx:= 6;
		tyP0931MagConv2.tyDC.tyBtnRemoteClamp.usiTxtIdx:= 6;
		tyP0931MagConv2.tyDC.tyBtnRemoteUnclamp.usiTxtIdx:= 6;

		tyP0931MagConv2.tyFB.tyBtnFixedClamp.usiTxtIdx:= 6;
		tyP0931MagConv2.tyFB.tyBtnFixedUnclamp.usiTxtIdx:= 6;
		tyP0931MagConv2.tyFB.tyBtnRemoteClamp.usiTxtIdx:= 6;
		tyP0931MagConv2.tyFB.tyBtnRemoteUnclamp.usiTxtIdx:= 6;

		tyP0931MagConv2.tyCom.tyBtnFixedUnclampRS.usiTxtIdx:= 5;
		tyP0931MagConv2.tyCom.tyBtnFixedClampRS.usiTxtIdx:= 10;
		tyP0931MagConv2.tyCom.tyBtnRemoteUnclampRS.usiTxtIdx:= 4;

	ELSE IF p_tyNtParamCurr.bMagAutoVerifyPrep = TRUE THEN

			tyP0931MagConv2.tyDC.tyBtnFixedClamp.usiTxtIdx:= 6;
			tyP0931MagConv2.tyDC.tyBtnFixedUnclamp.usiTxtIdx:= 6;
			tyP0931MagConv2.tyDC.tyBtnRemoteClamp.usiTxtIdx:= 6;
			tyP0931MagConv2.tyDC.tyBtnRemoteUnclamp.usiTxtIdx:= 6;

			tyP0931MagConv2.tyFB.tyBtnFixedClamp.usiTxtIdx:= 6;
			tyP0931MagConv2.tyFB.tyBtnFixedUnclamp.usiTxtIdx:= 6;
			tyP0931MagConv2.tyFB.tyBtnRemoteClamp.usiTxtIdx:= 6;
			tyP0931MagConv2.tyFB.tyBtnRemoteUnclamp.usiTxtIdx:= 6;

			tyP0931MagConv2.tyCom.tyBtnFixedUnclampRS.usiTxtIdx:= 5;
			tyP0931MagConv2.tyCom.tyBtnRemoteUnclampRS.usiTxtIdx:= 4;
		END_IF
	END_IF

	IF p_tyNtParamCurr.bMagAutoVerifyPrep AND p_tyNtParamCurr.bProjMagAWPrep = FALSE THEN
		tyP0931MagConv2.tyCom.tyBitmapMc.uiValueIdx	:= 0;
	ELSIF p_tyNtParamCurr.bMagAutoVerifyPrep AND p_tyNtParamCurr.bProjMagAWPrep THEN
		tyP0931MagConv2.tyCom.tyBitmapMc.uiValueIdx	:= 3;
	ELSIF p_tyNtParamCurr.bMagAutoVerifyPrep = FALSE AND p_tyNtParamCurr.bProjMagAWPrep = FALSE AND p_tyNtParamCurr.bProjMagSafetyBarPrep THEN
		tyP0931MagConv2.tyCom.tyBitmapMc.uiValueIdx	:= 203;
	ELSE
		tyP0931MagConv2.tyCom.tyBitmapMc.uiValueIdx	:= 234;
	END_IF

END_ACTION
```

#### Act_Main_P0932.st
```iecst
ACTION Act_Main_P0932:

	//Display
	tyP0932MagConv3.tyCom.tyBtnMagAIVPosSen1.uiRtStat.0			:= p_tyNtParamCurr.tyDISettings.diMag3AIVInPosSen1 = 0;
	tyP0932MagConv3.tyCom.tyBtnMagAIVPosSen2.uiRtStat.0			:= p_tyNtParamCurr.tyDISettings.diMag3AIVInPosSen2 = 0;
	tyP0932MagConv3.tyCom.tyBtnMagOrientationChkSen1.uiRtStat.0	:= p_tyNtParamCurr.tyDISettings.diMag3OrientChkSen1 = 0;
	tyP0932MagConv3.tyCom.tyBtnMagOrientationChkSen2.uiRtStat.0	:= p_tyNtParamCurr.tyDISettings.diMag3OrientChkSen2 = 0;

	//Hide the following when in MagAutoVerify
	tyP0932MagConv3.tyCom.tyBtnRemoteClampRS.uiRtStat.0			:= p_tyNtParamCurr.tyDISettings.diMag2RemoteClampRS = 0;
	tyP0932MagConv3.tyCom.tyBtnRemoteUnclampRS.uiRtStat.0		:=  p_tyNtParamCurr.tyDISettings.diMag3RemoteUnclampRS = 0 ;
	tyP0932MagConv3.tyCom.tyBtnFixedClampRS.uiRtStat.0			:= p_tyNtParamCurr.bMagAutoVerifyPrep;

//	tyP0932MagConv3.tyCom.tyBtnHeightSen.uiRtStat.0				:= NOT p_tyNtParamCurr.bMagAutoVerifyPrep;
	tyP0932MagConv3.tyCom.tyBtnCAB717Sen.uiRtStat.0				:= NOT p_tyNtParamCurr.bMagAutoVerifyPrep;
	tyP0932MagConv3.tyCom.tyBtnMagLargeSen.uiRtStat.0			:= NOT p_tyNtParamCurr.bMagAutoVerifyPrep;
	tyP0932MagConv3.tyCom.tyBtnMagSmallSen.uiRtStat.0			:= NOT p_tyNtParamCurr.bMagAutoVerifyPrep;
	tyP0932MagConv3.tyCom.tyBtnSelClampRS.uiRtStat.0			:= NOT p_tyNtParamCurr.bMagAutoVerifyPrep;
	tyP0932MagConv3.tyCom.tyBtnSelUnclampRS.uiRtStat.0			:= NOT p_tyNtParamCurr.bMagAutoVerifyPrep;
	tyP0932MagConv3.tyCom.tyBtnMagDetectSen.uiRtStat.0			:= NOT p_tyNtParamCurr.bProjFixClprMagDetectSenPrep;

	tyP0932MagConv3.tyCom.tyBtnHeightSen.uiRtStat.0				:= NOT p_tyNtParamCurr.bProjMagHeightChkPrep;

	IF p_tyNtParamCurr.bMagAutoVerifyPrep = FALSE THEN
		tyP0932MagConv3.tyDC.tyBtnFixedClamp.usiTxtIdx:= 6;
		tyP0932MagConv3.tyDC.tyBtnFixedUnclamp.usiTxtIdx:= 6;
		tyP0932MagConv3.tyDC.tyBtnRemoteClamp.usiTxtIdx:= 6;
		tyP0932MagConv3.tyDC.tyBtnRemoteUnclamp.usiTxtIdx:= 6;

		tyP0932MagConv3.tyFB.tyBtnFixedClamp.usiTxtIdx:= 6;
		tyP0932MagConv3.tyFB.tyBtnFixedUnclamp.usiTxtIdx:= 6;
		tyP0932MagConv3.tyFB.tyBtnRemoteClamp.usiTxtIdx:= 6;
		tyP0932MagConv3.tyFB.tyBtnRemoteUnclamp.usiTxtIdx:= 6;

		tyP0932MagConv3.tyCom.tyBtnFixedUnclampRS.usiTxtIdx:= 5;
		tyP0932MagConv3.tyCom.tyBtnFixedClampRS.usiTxtIdx:= 10;
		tyP0932MagConv3.tyCom.tyBtnRemoteUnclampRS.usiTxtIdx:= 4;

	ELSE IF p_tyNtParamCurr.bMagAutoVerifyPrep = TRUE THEN

			tyP0932MagConv3.tyDC.tyBtnFixedClamp.usiTxtIdx:= 6;
			tyP0932MagConv3.tyDC.tyBtnFixedUnclamp.usiTxtIdx:= 6;
			tyP0932MagConv3.tyDC.tyBtnRemoteClamp.usiTxtIdx:= 6;
			tyP0932MagConv3.tyDC.tyBtnRemoteUnclamp.usiTxtIdx:= 6;

			tyP0932MagConv3.tyFB.tyBtnFixedClamp.usiTxtIdx:= 6;
			tyP0932MagConv3.tyFB.tyBtnFixedUnclamp.usiTxtIdx:= 6;
			tyP0932MagConv3.tyFB.tyBtnRemoteClamp.usiTxtIdx:= 6;
			tyP0932MagConv3.tyFB.tyBtnRemoteUnclamp.usiTxtIdx:= 6;

			tyP0932MagConv3.tyCom.tyBtnFixedUnclampRS.usiTxtIdx:= 5;
			tyP0932MagConv3.tyCom.tyBtnRemoteUnclampRS.usiTxtIdx:= 4;
		END_IF
	END_IF

	IF p_tyNtParamCurr.bMagAutoVerifyPrep AND p_tyNtParamCurr.bProjMagAWPrep = FALSE THEN
		tyP0932MagConv3.tyCom.tyBitmapMc.uiValueIdx	:= 0;
	ELSIF p_tyNtParamCurr.bMagAutoVerifyPrep AND p_tyNtParamCurr.bProjMagAWPrep THEN
		tyP0932MagConv3.tyCom.tyBitmapMc.uiValueIdx	:= 3;
	ELSIF p_tyNtParamCurr.bMagAutoVerifyPrep = FALSE AND p_tyNtParamCurr.bProjMagAWPrep = FALSE AND p_tyNtParamCurr.bProjMagSafetyBarPrep THEN
		tyP0932MagConv3.tyCom.tyBitmapMc.uiValueIdx	:= 205;
	ELSE
		tyP0932MagConv3.tyCom.tyBitmapMc.uiValueIdx	:= 235;
	END_IF

END_ACTION
```
